LIN {X 0,Y 270.398,Z 235.226,A -85,B 0,C 180,E1 -18840.758,E2 -18840.758} C_VEL
LIN {X 0,Y 266.71,Z 211.064,A -85,B 0,C 180,E1 -18842.032,E2 -18842.032} C_VEL
LIN {X 0,Y 265.559,Z 205.31,A -85,B 0,C 180,E1 -18842.384,E2 -18842.384} C_VEL
LIN {X 0,Y 258.994,Z 190.687,A -85,B 0,C 180,E1 -18843.868,E2 -18843.868} C_VEL
LIN {X 0,Y 254.466,Z 181.608,A -85,B 0,C 180,E1 -18844.919,E2 -18844.919} C_VEL
LIN {X 0,Y 253.32,Z 178.871,A -85,B 0,C 180,E1 -18845.269,E2 -18845.269} C_VEL
LIN {X 0,Y 251.431,Z 171.126,A -85,B 0,C 180,E1 -18848.495,E2 -18848.495} C_VEL
LIN {X 0,Y 249.031,Z 162.462,A -85,B 0,C 180,E1 -18852.416,E2 -18852.416} C_VEL
LIN {X 0,Y 248.994,Z 162.469,A -85,B 0,C 180,E1 -18857.213,E2 -18857.213} C_VEL
LIN {X 0,Y 249.024,Z 162.467,A -85,B 0,C 180,E1 -18861.619,E2 -18861.619} C_VEL
LIN {X 0,Y 249.046,Z 162.465,A -85,B 0,C 180,E1 -18865.64,E2 -18865.64} C_VEL
LIN {X 0,Y 249.005,Z 162.467,A -85,B 0,C 180,E1 -18869.467,E2 -18869.467} C_VEL
LIN {X 0,Y 249.038,Z 162.464,A -85,B 0,C 180,E1 -18873.158,E2 -18873.158} C_VEL
LIN {X 0,Y 249.054,Z 162.46,A -85,B 0,C 180,E1 -18876.73,E2 -18876.73} C_VEL
LIN {X 0,Y 249.044,Z 162.449,A -85,B 0,C 180,E1 -18880.206,E2 -18880.206} C_VEL
LIN {X 0,Y 249.161,Z 162.447,A -85,B 0,C 180,E1 -18883.616,E2 -18883.616} C_VEL
LIN {X 0,Y 249.218,Z 162.442,A -85,B 0,C 180,E1 -18888.615,E2 -18888.615} C_VEL
LIN {X 0,Y 249.405,Z 162.403,A -85,B 0,C 180,E1 -18891.9,E2 -18891.9} C_VEL
LIN {X 0,Y 249.253,Z 162.436,A -85,B 0,C 180,E1 -18895.148,E2 -18895.148} C_VEL
LIN {X 0,Y 249.648,Z 162.378,A -85,B 0,C 180,E1 -18898.387,E2 -18898.387} C_VEL
LIN {X 0,Y 249.656,Z 162.378,A -85,B 0,C 180,E1 -18901.613,E2 -18901.613} C_VEL
LIN {X 0,Y 249.423,Z 162.413,A -85,B 0,C 180,E1 -18906.55,E2 -18906.55} C_VEL
LIN {X 0,Y 249.346,Z 162.414,A -85,B 0,C 180,E1 -18909.737,E2 -18909.737} C_VEL
LIN {X 0,Y 249.174,Z 162.433,A -85,B 0,C 180,E1 -18914.706,E2 -18914.706} C_VEL
LIN {X 0,Y 249.098,Z 162.452,A -85,B 0,C 180,E1 -18918.081,E2 -18918.081} C_VEL
LIN {X 0,Y 249.049,Z 162.463,A -85,B 0,C 180,E1 -18921.522,E2 -18921.522} C_VEL
LIN {X 0,Y 249.09,Z 162.452,A -85,B 0,C 180,E1 -18925.46,E2 -18925.46} C_VEL
LIN {X 0,Y 249.043,Z 162.455,A -85,B 0,C 180,E1 -18928.975,E2 -18928.975} C_VEL
LIN {X 0,Y 249.031,Z 162.458,A -85,B 0,C 180,E1 -18932.426,E2 -18932.426} C_VEL
LIN {X 0,Y 249.034,Z 162.457,A -85,B 0,C 180,E1 -18936.345,E2 -18936.345} C_VEL
LIN {X 0,Y 248.996,Z 162.444,A -85,B 0,C 180,E1 -18940.481,E2 -18940.481} C_VEL
LIN {X 0,Y 249.013,Z 162.453,A -85,B 0,C 180,E1 -18942.792,E2 -18942.792} C_VEL
LIN {X 0,Y 249.02,Z 162.464,A -85,B 0,C 180,E1 -18947.362,E2 -18947.362} C_VEL
LIN {X 0,Y 249.001,Z 162.471,A -85,B 0,C 180,E1 -18949.121,E2 -18949.121} C_VEL
LIN {X 0,Y 249.95,Z 165.205,A -85,B 0,C 180,E1 -18949.392,E2 -18949.392} C_VEL
LIN {X 0,Y 251.706,Z 167.591,A -85,B 0,C 180,E1 -18949.79,E2 -18949.79} C_VEL
LIN {X 0,Y 260.09,Z 181.406,A -85,B 0,C 180,E1 -18951.672,E2 -18951.672} C_VEL
LIN {X 0,Y 267.579,Z 196.726,A -85,B 0,C 180,E1 -18953.313,E2 -18953.313} C_VEL
LIN {X 0,Y 271.539,Z 205.911,A -85,B 0,C 180,E1 -18954.166,E2 -18954.166} C_VEL
LIN {X 0,Y 269.168,Z 267.873,A -85,B 0,C 180,E1 -18955.806,E2 -18955.806} C_VEL
LIN {X 0,Y 268.098,Z 281.069,A -85,B 0,C 180,E1 -18956.441,E2 -18956.441} C_VEL
LIN {X 0,Y 266.619,Z 293.102,A -85,B 0,C 180,E1 -18957.291,E2 -18957.291} C_VEL
LIN {X 0,Y 264.901,Z 304.551,A -85,B 0,C 180,E1 -18958.399,E2 -18958.399} C_VEL
LIN {X 0,Y 262.647,Z 316.276,A -85,B 0,C 180,E1 -18959.885,E2 -18959.885} C_VEL
LIN {X 0,Y 260.185,Z 326.779,A -85,B 0,C 180,E1 -18961.569,E2 -18961.569} C_VEL
LIN {X 0,Y 258.084,Z 335.342,A -85,B 0,C 180,E1 -18963.299,E2 -18963.299} C_VEL
LIN {X 0,Y 255.942,Z 343.505,A -85,B 0,C 180,E1 -18965.332,E2 -18965.332} C_VEL
LIN {X 0,Y 253.727,Z 350.862,A -85,B 0,C 180,E1 -18967.612,E2 -18967.612} C_VEL
LIN {X 0,Y 251.511,Z 357.887,A -85,B 0,C 180,E1 -18970.407,E2 -18970.407} C_VEL
LIN {X 0,Y 249.934,Z 362.747,A -85,B 0,C 180,E1 -18972.954,E2 -18972.954} C_VEL
LIN {X 0,Y 248.859,Z 366.06,A -85,B 0,C 180,E1 -18975.274,E2 -18975.274} C_VEL
LIN {X 0,Y 248.197,Z 367.857,A -85,B 0,C 180,E1 -18976.906,E2 -18976.906} C_VEL
LIN {X 0,Y 247.456,Z 370.137,A -85,B 0,C 180,E1 -18980.187,E2 -18980.187} C_VEL
LIN {X 0,Y 247.288,Z 370.694,A -85,B 0,C 180,E1 -18981.829,E2 -18981.829} C_VEL
LIN {X 0,Y 247.235,Z 370.759,A -85,B 0,C 180,E1 -18984.229,E2 -18984.229} C_VEL
LIN {X 0,Y 247.141,Z 369.941,A -85,B 0,C 180,E1 -18986.738,E2 -18986.738} C_VEL
LIN {X 0,Y 247.152,Z 368.924,A -85,B 0,C 180,E1 -18988.369,E2 -18988.369} C_VEL
LIN {X 0,Y 247.262,Z 367.49,A -85,B 0,C 180,E1 -18989.999,E2 -18989.999} C_VEL
LIN {X 0,Y 247.779,Z 364.536,A -85,B 0,C 180,E1 -18992.437,E2 -18992.437} C_VEL
LIN {X 0,Y 248.415,Z 360.557,A -85,B 0,C 180,E1 -18994.867,E2 -18994.867} C_VEL
LIN {X 0,Y 249.433,Z 355.427,A -85,B 0,C 180,E1 -18997.283,E2 -18997.283} C_VEL
LIN {X 0,Y 250.574,Z 348.992,A -85,B 0,C 180,E1 -18999.687,E2 -18999.687} C_VEL
LIN {X 0,Y 252.341,Z 340.966,A -85,B 0,C 180,E1 -19002.055,E2 -19002.055} C_VEL
LIN {X 0,Y 253.91,Z 332.787,A -85,B 0,C 180,E1 -19004.014,E2 -19004.014} C_VEL
LIN {X 0,Y 255.731,Z 322.787,A -85,B 0,C 180,E1 -19005.95,E2 -19005.95} C_VEL
LIN {X 0,Y 257.53,Z 311.457,A -85,B 0,C 180,E1 -19007.672,E2 -19007.672} C_VEL
LIN {X 0,Y 259.116,Z 300.335,A -85,B 0,C 180,E1 -19008.993,E2 -19008.993} C_VEL
LIN {X 0,Y 260.379,Z 287.896,A -85,B 0,C 180,E1 -19010.128,E2 -19010.128} C_VEL
LIN {X 0,Y 261.415,Z 274.564,A -85,B 0,C 180,E1 -19010.969,E2 -19010.969} C_VEL
LIN {X 0,Y 262.065,Z 261.42,A -85,B 0,C 180,E1 -19011.481,E2 -19011.481} C_VEL
LIN {X 0,Y 264.04,Z 197.022,A -85,B 0,C 180,E1 -19013.187,E2 -19013.187} C_VEL
LIN {X 0,Y 258.122,Z 181.409,A -85,B 0,C 180,E1 -19014.316,E2 -19014.316} C_VEL
LIN {X 0,Y 251.947,Z 168.721,A -85,B 0,C 180,E1 -19015.449,E2 -19015.449} C_VEL
LIN {X 0,Y 249.298,Z 163.437,A -85,B 0,C 180,E1 -19015.951,E2 -19015.951} C_VEL
LIN {X 0,Y 249.084,Z 162.459,A -85,B 0,C 180,E1 -19016.07,E2 -19016.07} C_VEL
LIN {X 0,Y 249.082,Z 162.456,A -85,B 0,C 180,E1 -19018.992,E2 -19018.992} C_VEL
LIN {X 0,Y 249.034,Z 162.462,A -85,B 0,C 180,E1 -19022.423,E2 -19022.423} C_VEL
LIN {X 0,Y 249.064,Z 162.458,A -85,B 0,C 180,E1 -19026.337,E2 -19026.337} C_VEL
LIN {X 0,Y 249.002,Z 162.466,A -85,B 0,C 180,E1 -19030.476,E2 -19030.476} C_VEL
LIN {X 0,Y 248.998,Z 162.467,A -85,B 0,C 180,E1 -19034.877,E2 -19034.877} C_VEL
LIN {X 0,Y 249.011,Z 162.463,A -85,B 0,C 180,E1 -19037.361,E2 -19037.361} C_VEL
LIN {X 0,Y 249.038,Z 162.46,A -85,B 0,C 180,E1 -19042.198,E2 -19042.198} C_VEL
LIN {X 0,Y 249.037,Z 162.464,A -85,B 0,C 180,E1 -19045.638,E2 -19045.638} C_VEL
LIN {X 0,Y 249.039,Z 162.465,A -85,B 0,C 180,E1 -19049.471,E2 -19049.471} C_VEL
LIN {X 0,Y 249.052,Z 162.456,A -85,B 0,C 180,E1 -19053.159,E2 -19053.159} C_VEL
LIN {X 0,Y 249.05,Z 162.46,A -85,B 0,C 180,E1 -19056.729,E2 -19056.729} C_VEL
LIN {X 0,Y 249.069,Z 162.458,A -85,B 0,C 180,E1 -19060.208,E2 -19060.208} C_VEL
LIN {X 0,Y 249.168,Z 162.441,A -85,B 0,C 180,E1 -19063.617,E2 -19063.617} C_VEL
LIN {X 0,Y 249.221,Z 162.439,A -85,B 0,C 180,E1 -19068.615,E2 -19068.615} C_VEL
LIN {X 0,Y 249.407,Z 162.4,A -85,B 0,C 180,E1 -19071.9,E2 -19071.9} C_VEL
LIN {X 0,Y 249.247,Z 162.411,A -85,B 0,C 180,E1 -19075.147,E2 -19075.147} C_VEL
LIN {X 0,Y 249.645,Z 162.383,A -85,B 0,C 180,E1 -19078.387,E2 -19078.387} C_VEL
LIN {X 0,Y 249.646,Z 162.385,A -85,B 0,C 180,E1 -19081.613,E2 -19081.613} C_VEL
LIN {X 0,Y 249.386,Z 162.415,A -85,B 0,C 180,E1 -19087.553,E2 -19087.553} C_VEL
LIN {X 0,Y 248.706,Z 162.507,A -85,B 0,C 180,E1 -19088.899,E2 -19088.899} C_VEL
LIN {X 0,Y 245.74,Z 162.873,A -85,B 0,C 180,E1 -19091.09,E2 -19091.09} C_VEL
LIN {X 0,Y 243.227,Z 163.188,A -85,B 0,C 180,E1 -19092.875,E2 -19092.875} C_VEL
LIN {X 0,Y 242.172,Z 163.32,A -85,B 0,C 180,E1 -19094.263,E2 -19094.263} C_VEL
LIN {X 0,Y 242.099,Z 163.326,A -85,B 0,C 180,E1 -19094.734,E2 -19094.734} C_VEL
LIN {X 0,Y 242.033,Z 163.341,A -85,B 0,C 180,E1 -19098.627,E2 -19098.627} C_VEL
LIN {X 0,Y 241.995,Z 163.343,A -85,B 0,C 180,E1 -19102.182,E2 -19102.182} C_VEL
LIN {X 0,Y 242.059,Z 163.334,A -85,B 0,C 180,E1 -19105.839,E2 -19105.839} C_VEL
LIN {X 0,Y 241.996,Z 163.342,A -85,B 0,C 180,E1 -19109.585,E2 -19109.585} C_VEL
LIN {X 0,Y 241.973,Z 163.345,A -85,B 0,C 180,E1 -19113.494,E2 -19113.494} C_VEL
LIN {X 0,Y 241.982,Z 163.344,A -85,B 0,C 180,E1 -19117.583,E2 -19117.583} C_VEL
LIN {X 0,Y 241.931,Z 163.351,A -85,B 0,C 180,E1 -19121.924,E2 -19121.924} C_VEL
LIN {X 0,Y 241.928,Z 163.347,A -85,B 0,C 180,E1 -19126.573,E2 -19126.573} C_VEL
LIN {X 0,Y 241.952,Z 163.347,A -85,B 0,C 180,E1 -19130.283,E2 -19130.283} C_VEL
LIN {X 0,Y 242.037,Z 163.517,A -85,B 0,C 180,E1 -19132.235,E2 -19132.235} C_VEL
LIN {X 0,Y 244.204,Z 172.335,A -85,B 0,C 180,E1 -19135.78,E2 -19135.78} C_VEL
LIN {X 0,Y 245.763,Z 179.777,A -85,B 0,C 180,E1 -19138.518,E2 -19138.518} C_VEL
LIN {X 0,Y 251.548,Z 194.496,A -85,B 0,C 180,E1 -19139.711,E2 -19139.711} C_VEL
LIN {X 0,Y 254.766,Z 216.953,A -85,B 0,C 180,E1 -19140.788,E2 -19140.788} C_VEL
LIN {X 0,Y 256.54,Z 232.58,A -85,B 0,C 180,E1 -19141.465,E2 -19141.465} C_VEL
LIN {X 0,Y 254.785,Z 288.121,A -85,B 0,C 180,E1 -19143.004,E2 -19143.004} C_VEL
LIN {X 0,Y 253.886,Z 301.362,A -85,B 0,C 180,E1 -19143.659,E2 -19143.659} C_VEL
LIN {X 0,Y 252.596,Z 312.538,A -85,B 0,C 180,E1 -19144.455,E2 -19144.455} C_VEL
LIN {X 0,Y 250.923,Z 324.371,A -85,B 0,C 180,E1 -19145.601,E2 -19145.601} C_VEL
LIN {X 0,Y 249.17,Z 335.145,A -85,B 0,C 180,E1 -19146.963,E2 -19146.963} C_VEL
LIN {X 0,Y 247.068,Z 346.126,A -85,B 0,C 180,E1 -19148.737,E2 -19148.737} C_VEL
LIN {X 0,Y 245.138,Z 356.346,A -85,B 0,C 180,E1 -19150.838,E2 -19150.838} C_VEL
LIN {X 0,Y 243.792,Z 364.08,A -85,B 0,C 180,E1 -19152.815,E2 -19152.815} C_VEL
LIN {X 0,Y 242.455,Z 370.774,A -85,B 0,C 180,E1 -19154.879,E2 -19154.879} C_VEL
LIN {X 0,Y 241.155,Z 377.362,A -85,B 0,C 180,E1 -19157.377,E2 -19157.377} C_VEL
LIN {X 0,Y 240.425,Z 382.612,A -85,B 0,C 180,E1 -19159.9,E2 -19159.9} C_VEL
LIN {X 0,Y 240.024,Z 386.683,A -85,B 0,C 180,E1 -19162.43,E2 -19162.43} C_VEL
LIN {X 0,Y 239.92,Z 389.691,A -85,B 0,C 180,E1 -19164.96,E2 -19164.96} C_VEL
LIN {X 0,Y 239.918,Z 391.144,A -85,B 0,C 180,E1 -19166.643,E2 -19166.643} C_VEL
LIN {X 0,Y 239.991,Z 392.169,A -85,B 0,C 180,E1 -19168.323,E2 -19168.323} C_VEL
LIN {X 0,Y 240.018,Z 392.796,A -85,B 0,C 180,E1 -19170.002,E2 -19170.002} C_VEL
LIN {X 0,Y 239.971,Z 393.027,A -85,B 0,C 180,E1 -19171.68,E2 -19171.68} C_VEL
LIN {X 0,Y 239.846,Z 392.272,A -85,B 0,C 180,E1 -19174.948,E2 -19174.948} C_VEL
LIN {X 0,Y 239.899,Z 391.228,A -85,B 0,C 180,E1 -19176.731,E2 -19176.731} C_VEL
LIN {X 0,Y 240.146,Z 389.843,A -85,B 0,C 180,E1 -19178.416,E2 -19178.416} C_VEL
LIN {X 0,Y 240.77,Z 386.934,A -85,B 0,C 180,E1 -19180.939,E2 -19180.939} C_VEL
LIN {X 0,Y 241.714,Z 383.006,A -85,B 0,C 180,E1 -19183.452,E2 -19183.452} C_VEL
LIN {X 0,Y 243.32,Z 377.97,A -85,B 0,C 180,E1 -19185.927,E2 -19185.927} C_VEL
LIN {X 0,Y 245.241,Z 371.662,A -85,B 0,C 180,E1 -19188.376,E2 -19188.376} C_VEL
LIN {X 0,Y 247.394,Z 363.783,A -85,B 0,C 180,E1 -19190.801,E2 -19190.801} C_VEL
LIN {X 0,Y 249.742,Z 355.777,A -85,B 0,C 180,E1 -19192.765,E2 -19192.765} C_VEL
LIN {X 0,Y 252.414,Z 346.028,A -85,B 0,C 180,E1 -19194.687,E2 -19194.687} C_VEL
LIN {X 0,Y 255.143,Z 335.198,A -85,B 0,C 180,E1 -19196.371,E2 -19196.371} C_VEL
LIN {X 0,Y 257.365,Z 324.63,A -85,B 0,C 180,E1 -19197.661,E2 -19197.661} C_VEL
LIN {X 0,Y 259.68,Z 311.918,A -85,B 0,C 180,E1 -19198.822,E2 -19198.822} C_VEL
LIN {X 0,Y 261.438,Z 299.188,A -85,B 0,C 180,E1 -19199.658,E2 -19199.658} C_VEL
LIN {X 0,Y 262.469,Z 286.951,A -85,B 0,C 180,E1 -19200.193,E2 -19200.193} C_VEL
LIN {X 0,Y 264.433,Z 236.333,A -85,B 0,C 180,E1 -19201.554,E2 -19201.554} C_VEL
LIN {X 0,Y 260.963,Z 213.15,A -85,B 0,C 180,E1 -19202.816,E2 -19202.816} C_VEL
LIN {X 0,Y 259.786,Z 207.659,A -85,B 0,C 180,E1 -19203.178,E2 -19203.178} C_VEL
LIN {X 0,Y 252.386,Z 191.247,A -85,B 0,C 180,E1 -19204.937,E2 -19204.937} C_VEL
LIN {X 0,Y 247.472,Z 181.709,A -85,B 0,C 180,E1 -19206.138,E2 -19206.138} C_VEL
LIN {X 0,Y 246.043,Z 178.541,A -85,B 0,C 180,E1 -19206.547,E2 -19206.547} C_VEL
LIN {X 0,Y 244.236,Z 171.448,A -85,B 0,C 180,E1 -19209.661,E2 -19209.661} C_VEL
LIN {X 0,Y 241.934,Z 163.348,A -85,B 0,C 180,E1 -19213.573,E2 -19213.573} C_VEL
LIN {X 0,Y 241.925,Z 163.351,A -85,B 0,C 180,E1 -19218.075,E2 -19218.075} C_VEL
LIN {X 0,Y 241.988,Z 163.343,A -85,B 0,C 180,E1 -19222.418,E2 -19222.418} C_VEL
LIN {X 0,Y 241.982,Z 163.344,A -85,B 0,C 180,E1 -19226.508,E2 -19226.508} C_VEL
LIN {X 0,Y 241.98,Z 163.345,A -85,B 0,C 180,E1 -19230.613,E2 -19230.613} C_VEL
LIN {X 0,Y 242.035,Z 163.333,A -85,B 0,C 180,E1 -19234.179,E2 -19234.179} C_VEL
LIN {X 0,Y 241.995,Z 163.34,A -85,B 0,C 180,E1 -19238.335,E2 -19238.335} C_VEL
LIN {X 0,Y 242.108,Z 163.326,A -85,B 0,C 180,E1 -19243.325,E2 -19243.325} C_VEL
LIN {X 0,Y 242.152,Z 163.321,A -85,B 0,C 180,E1 -19248.278,E2 -19248.278} C_VEL
LIN {X 0,Y 242.36,Z 163.28,A -85,B 0,C 180,E1 -19251.663,E2 -19251.663} C_VEL
LIN {X 0,Y 242.392,Z 163.289,A -85,B 0,C 180,E1 -19253.34,E2 -19253.34} C_VEL
LIN {X 0,Y 242.608,Z 163.254,A -85,B 0,C 180,E1 -19258.34,E2 -19258.34} C_VEL
LIN {X 0,Y 242.616,Z 163.254,A -85,B 0,C 180,E1 -19261.66,E2 -19261.66} C_VEL
LIN {X 0,Y 242.398,Z 163.289,A -85,B 0,C 180,E1 -19266.66,E2 -19266.66} C_VEL
LIN {X 0,Y 242.269,Z 163.299,A -85,B 0,C 180,E1 -19270.024,E2 -19270.024} C_VEL
LIN {X 0,Y 242.124,Z 163.313,A -85,B 0,C 180,E1 -19275.144,E2 -19275.144} C_VEL
LIN {X 0,Y 242.034,Z 163.327,A -85,B 0,C 180,E1 -19278.627,E2 -19278.627} C_VEL
LIN {X 0,Y 241.991,Z 163.341,A -85,B 0,C 180,E1 -19282.182,E2 -19282.182} C_VEL
LIN {X 0,Y 242.036,Z 163.334,A -85,B 0,C 180,E1 -19285.821,E2 -19285.821} C_VEL
LIN {X 0,Y 241.973,Z 163.338,A -85,B 0,C 180,E1 -19289.588,E2 -19289.588} C_VEL
LIN {X 0,Y 241.983,Z 163.337,A -85,B 0,C 180,E1 -19293.493,E2 -19293.493} C_VEL
LIN {X 0,Y 241.991,Z 163.34,A -85,B 0,C 180,E1 -19297.582,E2 -19297.582} C_VEL
LIN {X 0,Y 241.938,Z 163.324,A -85,B 0,C 180,E1 -19301.923,E2 -19301.923} C_VEL
LIN {X 0,Y 241.938,Z 163.35,A -85,B 0,C 180,E1 -19306.571,E2 -19306.571} C_VEL
LIN {X 0,Y 241.962,Z 163.343,A -85,B 0,C 180,E1 -19307.816,E2 -19307.816} C_VEL
LIN {X 0,Y 242.91,Z 166.061,A -85,B 0,C 180,E1 -19308.105,E2 -19308.105} C_VEL
LIN {X 0,Y 244.803,Z 168.669,A -85,B 0,C 180,E1 -19308.566,E2 -19308.566} C_VEL
LIN {X 0,Y 253.616,Z 182.897,A -85,B 0,C 180,E1 -19310.658,E2 -19310.658} C_VEL
LIN {X 0,Y 258.598,Z 192.44,A -85,B 0,C 180,E1 -19311.804,E2 -19311.804} C_VEL
LIN {X 0,Y 265.417,Z 207.578,A -85,B 0,C 180,E1 -19313.344,E2 -19313.344} C_VEL
LIN {X 0,Y 265.285,Z 215.569,A -85,B 0,C 180,E1 -19313.581,E2 -19313.581} C_VEL
LIN {X 0,Y 263.163,Z 268.09,A -85,B 0,C 180,E1 -19314.999,E2 -19314.999} C_VEL
LIN {X 0,Y 262.004,Z 281.688,A -85,B 0,C 180,E1 -19315.665,E2 -19315.665} C_VEL
LIN {X 0,Y 260.461,Z 293.792,A -85,B 0,C 180,E1 -19316.544,E2 -19316.544} C_VEL
LIN {X 0,Y 258.721,Z 304.882,A -85,B 0,C 180,E1 -19317.644,E2 -19317.644} C_VEL
LIN {X 0,Y 256.473,Z 316.095,A -85,B 0,C 180,E1 -19319.082,E2 -19319.082} C_VEL
LIN {X 0,Y 253.93,Z 326.686,A -85,B 0,C 180,E1 -19320.802,E2 -19320.802} C_VEL
LIN {X 0,Y 251.679,Z 335.319,A -85,B 0,C 180,E1 -19322.563,E2 -19322.563} C_VEL
LIN {X 0,Y 249.574,Z 342.981,A -85,B 0,C 180,E1 -19324.487,E2 -19324.487} C_VEL
LIN {X 0,Y 247.54,Z 349.798,A -85,B 0,C 180,E1 -19326.578,E2 -19326.578} C_VEL
LIN {X 0,Y 245.375,Z 356.227,A -85,B 0,C 180,E1 -19329.02,E2 -19329.02} C_VEL
LIN {X 0,Y 243.658,Z 361.302,A -85,B 0,C 180,E1 -19331.5,E2 -19331.5} C_VEL
LIN {X 0,Y 242.263,Z 365.227,A -85,B 0,C 180,E1 -19334.001,E2 -19334.001} C_VEL
LIN {X 0,Y 241.24,Z 368.108,A -85,B 0,C 180,E1 -19336.521,E2 -19336.521} C_VEL
LIN {X 0,Y 240.407,Z 370.424,A -85,B 0,C 180,E1 -19339.896,E2 -19339.896} C_VEL
LIN {X 0,Y 240.172,Z 371.171,A -85,B 0,C 180,E1 -19343.277,E2 -19343.277} C_VEL
LIN {X 0,Y 240.077,Z 370.927,A -85,B 0,C 180,E1 -19344.96,E2 -19344.96} C_VEL
LIN {X 0,Y 240.055,Z 370.304,A -85,B 0,C 180,E1 -19346.642,E2 -19346.642} C_VEL
LIN {X 0,Y 240.077,Z 369.302,A -85,B 0,C 180,E1 -19348.321,E2 -19348.321} C_VEL
LIN {X 0,Y 240.18,Z 367.899,A -85,B 0,C 180,E1 -19349.998,E2 -19349.998} C_VEL
LIN {X 0,Y 240.692,Z 364.974,A -85,B 0,C 180,E1 -19352.509,E2 -19352.509} C_VEL
LIN {X 0,Y 241.358,Z 361.028,A -85,B 0,C 180,E1 -19355.01,E2 -19355.01} C_VEL
LIN {X 0,Y 242.423,Z 355.942,A -85,B 0,C 180,E1 -19357.494,E2 -19357.494} C_VEL
LIN {X 0,Y 243.608,Z 349.555,A -85,B 0,C 180,E1 -19359.966,E2 -19359.966} C_VEL
LIN {X 0,Y 245.437,Z 341.577,A -85,B 0,C 180,E1 -19362.4,E2 -19362.4} C_VEL
LIN {X 0,Y 247.078,Z 333.455,A -85,B 0,C 180,E1 -19364.41,E2 -19364.41} C_VEL
LIN {X 0,Y 248.946,Z 323.547,A -85,B 0,C 180,E1 -19366.396,E2 -19366.396} C_VEL
LIN {X 0,Y 250.823,Z 312.331,A -85,B 0,C 180,E1 -19368.161,E2 -19368.161} C_VEL
LIN {X 0,Y 252.476,Z 301.338,A -85,B 0,C 180,E1 -19369.512,E2 -19369.512} C_VEL
LIN {X 0,Y 253.792,Z 289.172,A -85,B 0,C 180,E1 -19370.674,E2 -19370.674} C_VEL
LIN {X 0,Y 254.859,Z 276.299,A -85,B 0,C 180,E1 -19371.535,E2 -19371.535} C_VEL
LIN {X 0,Y 255.591,Z 262.578,A -85,B 0,C 180,E1 -19372.107,E2 -19372.107} C_VEL
LIN {X 0,Y 257.602,Z 198.497,A -85,B 0,C 180,E1 -19373.851,E2 -19373.851} C_VEL
LIN {X 0,Y 251.964,Z 183.792,A -85,B 0,C 180,E1 -19374.969,E2 -19374.969} C_VEL
LIN {X 0,Y 244.995,Z 169.7,A -85,B 0,C 180,E1 -19376.304,E2 -19376.304} C_VEL
LIN {X 0,Y 242.27,Z 164.505,A -85,B 0,C 180,E1 -19376.842,E2 -19376.842} C_VEL
LIN {X 0,Y 242.031,Z 163.337,A -85,B 0,C 180,E1 -19376.936,E2 -19376.936} C_VEL
LIN {X 0,Y 242.029,Z 163.335,A -85,B 0,C 180,E1 -19379.578,E2 -19379.578} C_VEL
LIN {X 0,Y 241.989,Z 163.34,A -85,B 0,C 180,E1 -19383.489,E2 -19383.489} C_VEL
LIN {X 0,Y 241.995,Z 163.339,A -85,B 0,C 180,E1 -19387.578,E2 -19387.578} C_VEL
LIN {X 0,Y 241.933,Z 163.348,A -85,B 0,C 180,E1 -19391.92,E2 -19391.92} C_VEL
LIN {X 0,Y 241.929,Z 163.346,A -85,B 0,C 180,E1 -19396.57,E2 -19396.57} C_VEL
LIN {X 0,Y 241.951,Z 163.346,A -85,B 0,C 180,E1 -19400.279,E2 -19400.279} C_VEL
LIN {X 0,Y 241.982,Z 163.342,A -85,B 0,C 180,E1 -19404.488,E2 -19404.488} C_VEL
LIN {X 0,Y 241.965,Z 163.343,A -85,B 0,C 180,E1 -19408.478,E2 -19408.478} C_VEL
LIN {X 0,Y 241.984,Z 163.335,A -85,B 0,C 180,E1 -19412.309,E2 -19412.309} C_VEL
LIN {X 0,Y 242.03,Z 163.336,A -85,B 0,C 180,E1 -19416.013,E2 -19416.013} C_VEL
LIN {X 0,Y 242.008,Z 163.337,A -85,B 0,C 180,E1 -19419.605,E2 -19419.605} C_VEL
LIN {X 0,Y 242.107,Z 163.323,A -85,B 0,C 180,E1 -19423.315,E2 -19423.315} C_VEL
LIN {X 0,Y 242.155,Z 163.319,A -85,B 0,C 180,E1 -19428.278,E2 -19428.278} C_VEL
LIN {X 0,Y 242.361,Z 163.277,A -85,B 0,C 180,E1 -19431.663,E2 -19431.663} C_VEL
LIN {X 0,Y 242.385,Z 163.26,A -85,B 0,C 180,E1 -19433.34,E2 -19433.34} C_VEL
LIN {X 0,Y 242.605,Z 163.259,A -85,B 0,C 180,E1 -19438.34,E2 -19438.34} C_VEL
LIN {X 0,Y 242.606,Z 163.262,A -85,B 0,C 180,E1 -19441.66,E2 -19441.66} C_VEL
LIN {X 0,Y 242.345,Z 163.293,A -85,B 0,C 180,E1 -19447.548,E2 -19447.548} C_VEL
LIN {X 0,Y 242.252,Z 163.309,A -85,B 0,C 180,E1 -19450.024,E2 -19450.024} C_VEL
LIN {X 0,Y 242.099,Z 163.326,A -85,B 0,C 180,E1 -19454.734,E2 -19454.734} C_VEL
LIN {X 0,Y 241.466,Z 163.409,A -85,B 0,C 180,E1 -19456.122,E2 -19456.122} C_VEL
LIN {X 0,Y 238.616,Z 163.766,A -85,B 0,C 180,E1 -19458.384,E2 -19458.384} C_VEL
LIN {X 0,Y 236.151,Z 164.072,A -85,B 0,C 180,E1 -19460.228,E2 -19460.228} C_VEL
LIN {X 0,Y 235.062,Z 164.206,A -85,B 0,C 180,E1 -19461.659,E2 -19461.659} C_VEL
LIN {X 0,Y 234.958,Z 164.219,A -85,B 0,C 180,E1 -19462.145,E2 -19462.145} C_VEL
LIN {X 0,Y 234.956,Z 164.223,A -85,B 0,C 180,E1 -19466.659,E2 -19466.659} C_VEL
LIN {X 0,Y 234.913,Z 164.228,A -85,B 0,C 180,E1 -19470.57,E2 -19470.57} C_VEL
LIN {X 0,Y 234.923,Z 164.226,A -85,B 0,C 180,E1 -19474.639,E2 -19474.639} C_VEL
LIN {X 0,Y 234.935,Z 164.222,A -85,B 0,C 180,E1 -19478.946,E2 -19478.946} C_VEL
LIN {X 0,Y 234.881,Z 164.228,A -85,B 0,C 180,E1 -19483.487,E2 -19483.487} C_VEL
LIN {X 0,Y 234.881,Z 164.225,A -85,B 0,C 180,E1 -19486.516,E2 -19486.516} C_VEL
LIN {X 0,Y 234.963,Z 164.296,A -85,B 0,C 180,E1 -19491.451,E2 -19491.451} C_VEL
LIN {X 0,Y 237.196,Z 173.334,A -85,B 0,C 180,E1 -19495.227,E2 -19495.227} C_VEL
LIN {X 0,Y 238.472,Z 179.327,A -85,B 0,C 180,E1 -19497.529,E2 -19497.529} C_VEL
LIN {X 0,Y 245.438,Z 196.678,A -85,B 0,C 180,E1 -19499.029,E2 -19499.029} C_VEL
LIN {X 0,Y 248.322,Z 216.781,A -85,B 0,C 180,E1 -19500.032,E2 -19500.032} C_VEL
LIN {X 0,Y 250.179,Z 234.602,A -85,B 0,C 180,E1 -19500.816,E2 -19500.816} C_VEL
LIN {X 0,Y 248.329,Z 288.491,A -85,B 0,C 180,E1 -19502.347,E2 -19502.347} C_VEL
LIN {X 0,Y 247.366,Z 301.6,A -85,B 0,C 180,E1 -19503.021,E2 -19503.021} C_VEL
LIN {X 0,Y 246.047,Z 312.647,A -85,B 0,C 180,E1 -19503.838,E2 -19503.838} C_VEL
LIN {X 0,Y 244.462,Z 323.498,A -85,B 0,C 180,E1 -19504.912,E2 -19504.912} C_VEL
LIN {X 0,Y 242.616,Z 334.378,A -85,B 0,C 180,E1 -19506.303,E2 -19506.303} C_VEL
LIN {X 0,Y 240.73,Z 344.388,A -85,B 0,C 180,E1 -19507.923,E2 -19507.923} C_VEL
LIN {X 0,Y 238.784,Z 353.578,A -85,B 0,C 180,E1 -19509.769,E2 -19509.769} C_VEL
LIN {X 0,Y 237.184,Z 362.309,A -85,B 0,C 180,E1 -19511.961,E2 -19511.961} C_VEL
LIN {X 0,Y 235.549,Z 370.257,A -85,B 0,C 180,E1 -19514.425,E2 -19514.425} C_VEL
LIN {X 0,Y 234.203,Z 376.882,A -85,B 0,C 180,E1 -19516.995,E2 -19516.995} C_VEL
LIN {X 0,Y 233.411,Z 382.166,A -85,B 0,C 180,E1 -19519.594,E2 -19519.594} C_VEL
LIN {X 0,Y 232.974,Z 386.266,A -85,B 0,C 180,E1 -19522.2,E2 -19522.2} C_VEL
LIN {X 0,Y 232.842,Z 389.408,A -85,B 0,C 180,E1 -19524.912,E2 -19524.912} C_VEL
LIN {X 0,Y 232.819,Z 390.776,A -85,B 0,C 180,E1 -19526.54,E2 -19526.54} C_VEL
LIN {X 0,Y 232.919,Z 391.816,A -85,B 0,C 180,E1 -19528.273,E2 -19528.273} C_VEL
LIN {X 0,Y 232.946,Z 392.455,A -85,B 0,C 180,E1 -19530.002,E2 -19530.002} C_VEL
LIN {X 0,Y 232.898,Z 392.698,A -85,B 0,C 180,E1 -19531.731,E2 -19531.731} C_VEL
LIN {X 0,Y 232.77,Z 392.081,A -85,B 0,C 180,E1 -19534.884,E2 -19534.884} C_VEL
LIN {X 0,Y 232.82,Z 390.946,A -85,B 0,C 180,E1 -19536.937,E2 -19536.937} C_VEL
LIN {X 0,Y 233.094,Z 389.574,A -85,B 0,C 180,E1 -19538.672,E2 -19538.672} C_VEL
LIN {X 0,Y 233.767,Z 386.69,A -85,B 0,C 180,E1 -19541.271,E2 -19541.271} C_VEL
LIN {X 0,Y 234.787,Z 382.791,A -85,B 0,C 180,E1 -19543.857,E2 -19543.857} C_VEL
LIN {X 0,Y 236.48,Z 377.785,A -85,B 0,C 180,E1 -19546.401,E2 -19546.401} C_VEL
LIN {X 0,Y 238.793,Z 370.492,A -85,B 0,C 180,E1 -19549.271,E2 -19549.271} C_VEL
LIN {X 0,Y 241.198,Z 362.198,A -85,B 0,C 180,E1 -19551.81,E2 -19551.81} C_VEL
LIN {X 0,Y 243.751,Z 353.944,A -85,B 0,C 180,E1 -19553.808,E2 -19553.808} C_VEL
LIN {X 0,Y 246.603,Z 343.874,A -85,B 0,C 180,E1 -19555.762,E2 -19555.762} C_VEL
LIN {X 0,Y 249.443,Z 332.483,A -85,B 0,C 180,E1 -19557.476,E2 -19557.476} C_VEL
LIN {X 0,Y 251.838,Z 321.323,A -85,B 0,C 180,E1 -19558.778,E2 -19558.778} C_VEL
LIN {X 0,Y 254.062,Z 308.847,A -85,B 0,C 180,E1 -19559.864,E2 -19559.864} C_VEL
LIN {X 0,Y 255.777,Z 295.518,A -85,B 0,C 180,E1 -19560.668,E2 -19560.668} C_VEL
LIN {X 0,Y 256.731,Z 282.506,A -85,B 0,C 180,E1 -19561.17,E2 -19561.17} C_VEL
LIN {X 0,Y 258.543,Z 237.621,A -85,B 0,C 180,E1 -19562.378,E2 -19562.378} C_VEL
LIN {X 0,Y 254.711,Z 211.904,A -85,B 0,C 180,E1 -19563.839,E2 -19563.839} C_VEL
LIN {X 0,Y 249.856,Z 200.467,A -85,B 0,C 180,E1 -19565.047,E2 -19565.047} C_VEL
LIN {X 0,Y 243.325,Z 186.984,A -85,B 0,C 180,E1 -19566.711,E2 -19566.711} C_VEL
LIN {X 0,Y 238.785,Z 178.173,A -85,B 0,C 180,E1 -19567.937,E2 -19567.937} C_VEL
LIN {X 0,Y 236.427,Z 169.538,A -85,B 0,C 180,E1 -19572,E2 -19572} C_VEL
LIN {X 0,Y 234.875,Z 164.228,A -85,B 0,C 180,E1 -19574.714,E2 -19574.714} C_VEL
LIN {X 0,Y 234.867,Z 164.229,A -85,B 0,C 180,E1 -19578.829,E2 -19578.829} C_VEL
LIN {X 0,Y 234.928,Z 164.222,A -85,B 0,C 180,E1 -19583.251,E2 -19583.251} C_VEL
LIN {X 0,Y 234.956,Z 164.218,A -85,B 0,C 180,E1 -19587.424,E2 -19587.424} C_VEL
LIN {X 0,Y 234.904,Z 164.222,A -85,B 0,C 180,E1 -19591.4,E2 -19591.4} C_VEL
LIN {X 0,Y 234.956,Z 164.218,A -85,B 0,C 180,E1 -19595.243,E2 -19595.243} C_VEL
LIN {X 0,Y 234.942,Z 164.213,A -85,B 0,C 180,E1 -19598.963,E2 -19598.963} C_VEL
LIN {X 0,Y 235.052,Z 164.205,A -85,B 0,C 180,E1 -19603.098,E2 -19603.098} C_VEL
LIN {X 0,Y 235.084,Z 164.199,A -85,B 0,C 180,E1 -19607.921,E2 -19607.921} C_VEL
LIN {X 0,Y 235.298,Z 164.159,A -85,B 0,C 180,E1 -19611.411,E2 -19611.411} C_VEL
LIN {X 0,Y 235.343,Z 164.166,A -85,B 0,C 180,E1 -19613.14,E2 -19613.14} C_VEL
LIN {X 0,Y 235.567,Z 164.13,A -85,B 0,C 180,E1 -19618.291,E2 -19618.291} C_VEL
LIN {X 0,Y 235.575,Z 164.131,A -85,B 0,C 180,E1 -19621.71,E2 -19621.71} C_VEL
LIN {X 0,Y 235.35,Z 164.166,A -85,B 0,C 180,E1 -19626.86,E2 -19626.86} C_VEL
LIN {X 0,Y 235.215,Z 164.181,A -85,B 0,C 180,E1 -19630.328,E2 -19630.328} C_VEL
LIN {X 0,Y 235.073,Z 164.195,A -85,B 0,C 180,E1 -19635.609,E2 -19635.609} C_VEL
LIN {X 0,Y 234.973,Z 164.203,A -85,B 0,C 180,E1 -19639.209,E2 -19639.209} C_VEL
LIN {X 0,Y 234.941,Z 164.216,A -85,B 0,C 180,E1 -19642.885,E2 -19642.885} C_VEL
LIN {X 0,Y 234.95,Z 164.22,A -85,B 0,C 180,E1 -19646.66,E2 -19646.66} C_VEL
LIN {X 0,Y 234.903,Z 164.225,A -85,B 0,C 180,E1 -19650.572,E2 -19650.572} C_VEL
LIN {X 0,Y 234.931,Z 164.222,A -85,B 0,C 180,E1 -19654.638,E2 -19654.638} C_VEL
LIN {X 0,Y 234.918,Z 164.216,A -85,B 0,C 180,E1 -19658.936,E2 -19658.936} C_VEL
LIN {X 0,Y 234.891,Z 164.222,A -85,B 0,C 180,E1 -19663.486,E2 -19663.486} C_VEL
LIN {X 0,Y 234.912,Z 164.225,A -85,B 0,C 180,E1 -19666.371,E2 -19666.371} C_VEL
LIN {X 0,Y 236.006,Z 167.195,A -85,B 0,C 180,E1 -19666.753,E2 -19666.753} C_VEL
LIN {X 0,Y 237.794,Z 169.484,A -85,B 0,C 180,E1 -19667.214,E2 -19667.214} C_VEL
LIN {X 0,Y 247.041,Z 184.175,A -85,B 0,C 180,E1 -19669.549,E2 -19669.549} C_VEL
LIN {X 0,Y 252.242,Z 193.63,A -85,B 0,C 180,E1 -19670.798,E2 -19670.798} C_VEL
LIN {X 0,Y 258.943,Z 208.37,A -85,B 0,C 180,E1 -19672.39,E2 -19672.39} C_VEL
LIN {X 0,Y 259.633,Z 210.013,A -85,B 0,C 180,E1 -19672.552,E2 -19672.552} C_VEL
LIN {X 0,Y 257.22,Z 268.266,A -85,B 0,C 180,E1 -19674.152,E2 -19674.152} C_VEL
LIN {X 0,Y 256.065,Z 281.47,A -85,B 0,C 180,E1 -19674.803,E2 -19674.803} C_VEL
LIN {X 0,Y 254.383,Z 294.248,A -85,B 0,C 180,E1 -19675.741,E2 -19675.741} C_VEL
LIN {X 0,Y 252.557,Z 305.347,A -85,B 0,C 180,E1 -19676.867,E2 -19676.867} C_VEL
LIN {X 0,Y 250.058,Z 317.212,A -85,B 0,C 180,E1 -19678.434,E2 -19678.434} C_VEL
LIN {X 0,Y 247.428,Z 327.665,A -85,B 0,C 180,E1 -19680.192,E2 -19680.192} C_VEL
LIN {X 0,Y 244.849,Z 337.039,A -85,B 0,C 180,E1 -19682.196,E2 -19682.196} C_VEL
LIN {X 0,Y 242.21,Z 346.06,A -85,B 0,C 180,E1 -19684.659,E2 -19684.659} C_VEL
LIN {X 0,Y 239.754,Z 353.307,A -85,B 0,C 180,E1 -19687.144,E2 -19687.144} C_VEL
LIN {X 0,Y 238.035,Z 358.185,A -85,B 0,C 180,E1 -19689.248,E2 -19689.248} C_VEL
LIN {X 0,Y 236.29,Z 363.047,A -85,B 0,C 180,E1 -19691.89,E2 -19691.89} C_VEL
LIN {X 0,Y 234.993,Z 366.504,A -85,B 0,C 180,E1 -19694.384,E2 -19694.384} C_VEL
LIN {X 0,Y 234.296,Z 368.354,A -85,B 0,C 180,E1 -19696.114,E2 -19696.114} C_VEL
LIN {X 0,Y 233.751,Z 369.736,A -85,B 0,C 180,E1 -19697.849,E2 -19697.849} C_VEL
LIN {X 0,Y 233.158,Z 371.298,A -85,B 0,C 180,E1 -19701.33,E2 -19701.33} C_VEL
LIN {X 0,Y 233.066,Z 371.378,A -85,B 0,C 180,E1 -19704.33,E2 -19704.33} C_VEL
LIN {X 0,Y 232.972,Z 370.666,A -85,B 0,C 180,E1 -19706.54,E2 -19706.54} C_VEL
LIN {X 0,Y 233.004,Z 369.679,A -85,B 0,C 180,E1 -19708.27,E2 -19708.27} C_VEL
LIN {X 0,Y 233.1,Z 368.302,A -85,B 0,C 180,E1 -19709.998,E2 -19709.998} C_VEL
LIN {X 0,Y 233.606,Z 365.404,A -85,B 0,C 180,E1 -19712.585,E2 -19712.585} C_VEL
LIN {X 0,Y 234.301,Z 361.492,A -85,B 0,C 180,E1 -19715.161,E2 -19715.161} C_VEL
LIN {X 0,Y 235.417,Z 356.448,A -85,B 0,C 180,E1 -19717.719,E2 -19717.719} C_VEL
LIN {X 0,Y 236.65,Z 350.115,A -85,B 0,C 180,E1 -19720.262,E2 -19720.262} C_VEL
LIN {X 0,Y 238.546,Z 342.186,A -85,B 0,C 180,E1 -19722.764,E2 -19722.764} C_VEL
LIN {X 0,Y 240.433,Z 333.265,A -85,B 0,C 180,E1 -19725.027,E2 -19725.027} C_VEL
LIN {X 0,Y 242.391,Z 323.178,A -85,B 0,C 180,E1 -19727.07,E2 -19727.07} C_VEL
LIN {X 0,Y 244.365,Z 311.787,A -85,B 0,C 180,E1 -19728.876,E2 -19728.876} C_VEL
LIN {X 0,Y 246.088,Z 300.589,A -85,B 0,C 180,E1 -19730.258,E2 -19730.258} C_VEL
LIN {X 0,Y 247.332,Z 289.235,A -85,B 0,C 180,E1 -19731.348,E2 -19731.348} C_VEL
LIN {X 0,Y 248.44,Z 276.221,A -85,B 0,C 180,E1 -19732.23,E2 -19732.23} C_VEL
LIN {X 0,Y 249.142,Z 263.734,A -85,B 0,C 180,E1 -19732.765,E2 -19732.765} C_VEL
LIN {X 0,Y 251.217,Z 200.011,A -85,B 0,C 180,E1 -19734.545,E2 -19734.545} C_VEL
LIN {X 0,Y 245.601,Z 185.524,A -85,B 0,C 180,E1 -19735.706,E2 -19735.706} C_VEL
LIN {X 0,Y 238.055,Z 170.745,A -85,B 0,C 180,E1 -19737.213,E2 -19737.213} C_VEL
LIN {X 0,Y 235.249,Z 165.47,A -85,B 0,C 180,E1 -19737.796,E2 -19737.796} C_VEL
LIN {X 0,Y 234.967,Z 164.217,A -85,B 0,C 180,E1 -19737.963,E2 -19737.963} C_VEL
LIN {X 0,Y 234.958,Z 164.215,A -85,B 0,C 180,E1 -19742.573,E2 -19742.573} C_VEL
LIN {X 0,Y 234.936,Z 164.217,A -85,B 0,C 180,E1 -19746.745,E2 -19746.745} C_VEL
LIN {X 0,Y 234.938,Z 164.216,A -85,B 0,C 180,E1 -19748.942,E2 -19748.942} C_VEL
LIN {X 0,Y 234.882,Z 164.227,A -85,B 0,C 180,E1 -19753.484,E2 -19753.484} C_VEL
LIN {X 0,Y 234.882,Z 164.223,A -85,B 0,C 180,E1 -19756.512,E2 -19756.512} C_VEL
LIN {X 0,Y 234.913,Z 164.222,A -85,B 0,C 180,E1 -19761.077,E2 -19761.077} C_VEL
LIN {X 0,Y 234.924,Z 164.223,A -85,B 0,C 180,E1 -19765.361,E2 -19765.361} C_VEL
LIN {X 0,Y 234.914,Z 164.224,A -85,B 0,C 180,E1 -19769.429,E2 -19769.429} C_VEL
LIN {X 0,Y 234.985,Z 164.212,A -85,B 0,C 180,E1 -19773.793,E2 -19773.793} C_VEL
LIN {X 0,Y 234.96,Z 164.209,A -85,B 0,C 180,E1 -19778.965,E2 -19778.965} C_VEL
LIN {X 0,Y 235.047,Z 164.204,A -85,B 0,C 180,E1 -19783.091,E2 -19783.091} C_VEL
LIN {X 0,Y 235.087,Z 164.2,A -85,B 0,C 180,E1 -19787.92,E2 -19787.92} C_VEL
LIN {X 0,Y 235.301,Z 164.157,A -85,B 0,C 180,E1 -19791.411,E2 -19791.411} C_VEL
LIN {X 0,Y 235.337,Z 164.137,A -85,B 0,C 180,E1 -19793.139,E2 -19793.139} C_VEL
LIN {X 0,Y 235.564,Z 164.136,A -85,B 0,C 180,E1 -19798.29,E2 -19798.29} C_VEL
LIN {X 0,Y 235.565,Z 164.139,A -85,B 0,C 180,E1 -19801.709,E2 -19801.709} C_VEL
LIN {X 0,Y 235.337,Z 164.169,A -85,B 0,C 180,E1 -19806.86,E2 -19806.86} C_VEL
LIN {X 0,Y 235.2,Z 164.188,A -85,B 0,C 180,E1 -19810.328,E2 -19810.328} C_VEL
LIN {X 0,Y 235.065,Z 164.203,A -85,B 0,C 180,E1 -19815.61,E2 -19815.61} C_VEL
LIN {X 0,Y 234.975,Z 164.217,A -85,B 0,C 180,E1 -19819.208,E2 -19819.208} C_VEL
LIN {X 0,Y 234.958,Z 164.219,A -85,B 0,C 180,E1 -19822.145,E2 -19822.145} C_VEL
LIN {X 0,Y 234.253,Z 164.308,A -85,B 0,C 180,E1 -19823.576,E2 -19823.576} C_VEL
LIN {X 0,Y 231.407,Z 164.662,A -85,B 0,C 180,E1 -19825.911,E2 -19825.911} C_VEL
LIN {X 0,Y 229.008,Z 164.961,A -85,B 0,C 180,E1 -19827.815,E2 -19827.815} C_VEL
LIN {X 0,Y 227.975,Z 165.089,A -85,B 0,C 180,E1 -19829.292,E2 -19829.292} C_VEL
LIN {X 0,Y 227.888,Z 165.1,A -85,B 0,C 180,E1 -19829.793,E2 -19829.793} C_VEL
LIN {X 0,Y 227.87,Z 165.103,A -85,B 0,C 180,E1 -19833.722,E2 -19833.722} C_VEL
LIN {X 0,Y 227.837,Z 165.108,A -85,B 0,C 180,E1 -19838.092,E2 -19838.092} C_VEL
LIN {X 0,Y 227.805,Z 165.11,A -85,B 0,C 180,E1 -19842.744,E2 -19842.744} C_VEL
LIN {X 0,Y 227.805,Z 165.101,A -85,B 0,C 180,E1 -19847.259,E2 -19847.259} C_VEL
LIN {X 0,Y 227.903,Z 165.238,A -85,B 0,C 180,E1 -19850.679,E2 -19850.679} C_VEL
LIN {X 0,Y 230.111,Z 174.09,A -85,B 0,C 180,E1 -19854.531,E2 -19854.531} C_VEL
LIN {X 0,Y 231.133,Z 178.748,A -85,B 0,C 180,E1 -19856.452,E2 -19856.452} C_VEL
LIN {X 0,Y 238.594,Z 196.868,A -85,B 0,C 180,E1 -19858.141,E2 -19858.141} C_VEL
LIN {X 0,Y 239.752,Z 200.592,A -85,B 0,C 180,E1 -19858.422,E2 -19858.422} C_VEL
LIN {X 0,Y 243.104,Z 227.268,A -85,B 0,C 180,E1 -19859.736,E2 -19859.736} C_VEL
LIN {X 0,Y 243.841,Z 235.23,A -85,B 0,C 180,E1 -19860.086,E2 -19860.086} C_VEL
LIN {X 0,Y 241.979,Z 287.705,A -85,B 0,C 180,E1 -19861.606,E2 -19861.606} C_VEL
LIN {X 0,Y 241.016,Z 300.321,A -85,B 0,C 180,E1 -19862.25,E2 -19862.25} C_VEL
LIN {X 0,Y 239.531,Z 312.756,A -85,B 0,C 180,E1 -19863.187,E2 -19863.187} C_VEL
LIN {X 0,Y 237.724,Z 324.397,A -85,B 0,C 180,E1 -19864.384,E2 -19864.384} C_VEL
LIN {X 0,Y 235.586,Z 336.321,A -85,B 0,C 180,E1 -19866.019,E2 -19866.019} C_VEL
LIN {X 0,Y 233.349,Z 346.964,A -85,B 0,C 180,E1 -19867.887,E2 -19867.887} C_VEL
LIN {X 0,Y 231.38,Z 356.575,A -85,B 0,C 180,E1 -19870.021,E2 -19870.021} C_VEL
LIN {X 0,Y 229.862,Z 364.453,A -85,B 0,C 180,E1 -19872.199,E2 -19872.199} C_VEL
LIN {X 0,Y 228.161,Z 372.124,A -85,B 0,C 180,E1 -19874.824,E2 -19874.824} C_VEL
LIN {X 0,Y 226.873,Z 378.294,A -85,B 0,C 180,E1 -19877.478,E2 -19877.478} C_VEL
LIN {X 0,Y 226.186,Z 383.198,A -85,B 0,C 180,E1 -19880.162,E2 -19880.162} C_VEL
LIN {X 0,Y 225.821,Z 386.962,A -85,B 0,C 180,E1 -19882.851,E2 -19882.851} C_VEL
LIN {X 0,Y 225.737,Z 389.295,A -85,B 0,C 180,E1 -19885.053,E2 -19885.053} C_VEL
LIN {X 0,Y 225.824,Z 391.461,A -85,B 0,C 180,E1 -19888.218,E2 -19888.218} C_VEL
LIN {X 0,Y 225.875,Z 392.114,A -85,B 0,C 180,E1 -19890.002,E2 -19890.002} C_VEL
LIN {X 0,Y 225.802,Z 392.368,A -85,B 0,C 180,E1 -19891.785,E2 -19891.785} C_VEL
LIN {X 0,Y 225.689,Z 391.868,A -85,B 0,C 180,E1 -19894.805,E2 -19894.805} C_VEL
LIN {X 0,Y 225.766,Z 390.665,A -85,B 0,C 180,E1 -19897.154,E2 -19897.154} C_VEL
LIN {X 0,Y 226.038,Z 389.304,A -85,B 0,C 180,E1 -19898.945,E2 -19898.945} C_VEL
LIN {X 0,Y 226.757,Z 386.447,A -85,B 0,C 180,E1 -19901.624,E2 -19901.624} C_VEL
LIN {X 0,Y 227.88,Z 382.576,A -85,B 0,C 180,E1 -19904.285,E2 -19904.285} C_VEL
LIN {X 0,Y 229.654,Z 377.599,A -85,B 0,C 180,E1 -19906.903,E2 -19906.903} C_VEL
LIN {X 0,Y 231.742,Z 371.358,A -85,B 0,C 180,E1 -19909.489,E2 -19909.489} C_VEL
LIN {X 0,Y 234.115,Z 363.593,A -85,B 0,C 180,E1 -19912.041,E2 -19912.041} C_VEL
LIN {X 0,Y 237.254,Z 353.895,A -85,B 0,C 180,E1 -19914.502,E2 -19914.502} C_VEL
LIN {X 0,Y 240.238,Z 343.897,A -85,B 0,C 180,E1 -19916.497,E2 -19916.497} C_VEL
LIN {X 0,Y 243.184,Z 332.6,A -85,B 0,C 180,E1 -19918.246,E2 -19918.246} C_VEL
LIN {X 0,Y 245.657,Z 321.545,A -85,B 0,C 180,E1 -19919.572,E2 -19919.572} C_VEL
LIN {X 0,Y 247.953,Z 309.281,A -85,B 0,C 180,E1 -19920.678,E2 -19920.678} C_VEL
LIN {X 0,Y 249.71,Z 296.328,A -85,B 0,C 180,E1 -19921.497,E2 -19921.497} C_VEL
LIN {X 0,Y 250.801,Z 282.551,A -85,B 0,C 180,E1 -19922.052,E2 -19922.052} C_VEL
LIN {X 0,Y 252.632,Z 238.145,A -85,B 0,C 180,E1 -19923.279,E2 -19923.279} C_VEL
LIN {X 0,Y 249.176,Z 214.438,A -85,B 0,C 180,E1 -19924.671,E2 -19924.671} C_VEL
LIN {X 0,Y 242.142,Z 198.532,A -85,B 0,C 180,E1 -19926.505,E2 -19926.505} C_VEL
LIN {X 0,Y 236.185,Z 186.665,A -85,B 0,C 180,E1 -19928.122,E2 -19928.122} C_VEL
LIN {X 0,Y 233.376,Z 181.576,A -85,B 0,C 180,E1 -19928.907,E2 -19928.907} C_VEL
LIN {X 0,Y 231.419,Z 177.697,A -85,B 0,C 180,E1 -19929.511,E2 -19929.511} C_VEL
LIN {X 0,Y 229.289,Z 170.138,A -85,B 0,C 180,E1 -19933.284,E2 -19933.284} C_VEL
LIN {X 0,Y 227.849,Z 165.103,A -85,B 0,C 180,E1 -19936.04,E2 -19936.04} C_VEL
LIN {X 0,Y 227.832,Z 165.106,A -85,B 0,C 180,E1 -19940.462,E2 -19940.462} C_VEL
LIN {X 0,Y 227.883,Z 165.101,A -85,B 0,C 180,E1 -19944.129,E2 -19944.129} C_VEL
LIN {X 0,Y 227.859,Z 165.104,A -85,B 0,C 180,E1 -19948.376,E2 -19948.376} C_VEL
LIN {X 0,Y 227.858,Z 165.101,A -85,B 0,C 180,E1 -19952.441,E2 -19952.441} C_VEL
LIN {X 0,Y 227.893,Z 165.095,A -85,B 0,C 180,E1 -19956.365,E2 -19956.365} C_VEL
LIN {X 0,Y 227.892,Z 165.083,A -85,B 0,C 180,E1 -19960.17,E2 -19960.17} C_VEL
LIN {X 0,Y 228.001,Z 165.081,A -85,B 0,C 180,E1 -19963.894,E2 -19963.894} C_VEL
LIN {X 0,Y 228.127,Z 165.067,A -85,B 0,C 180,E1 -19969.348,E2 -19969.348} C_VEL
LIN {X 0,Y 228.295,Z 165.04,A -85,B 0,C 180,E1 -19972.927,E2 -19972.927} C_VEL
LIN {X 0,Y 228.501,Z 165.01,A -85,B 0,C 180,E1 -19978.238,E2 -19978.238} C_VEL
LIN {X 0,Y 228.534,Z 165.007,A -85,B 0,C 180,E1 -19981.762,E2 -19981.762} C_VEL
LIN {X 0,Y 228.303,Z 165.04,A -85,B 0,C 180,E1 -19987.073,E2 -19987.073} C_VEL
LIN {X 0,Y 228.146,Z 165.064,A -85,B 0,C 180,E1 -19990.651,E2 -19990.651} C_VEL
LIN {X 0,Y 228.021,Z 165.08,A -85,B 0,C 180,E1 -19996.105,E2 -19996.105} C_VEL
LIN {X 0,Y 227.929,Z 165.094,A -85,B 0,C 180,E1 -20001.717,E2 -20001.717} C_VEL
LIN {X 0,Y 227.927,Z 165.094,A -85,B 0,C 180,E1 -20006.592,E2 -20006.592} C_VEL
LIN {X 0,Y 227.878,Z 165.098,A -85,B 0,C 180,E1 -20010.281,E2 -20010.281} C_VEL
LIN {X 0,Y 227.88,Z 165.095,A -85,B 0,C 180,E1 -20013.72,E2 -20013.72} C_VEL
LIN {X 0,Y 227.847,Z 165.103,A -85,B 0,C 180,E1 -20018.091,E2 -20018.091} C_VEL
LIN {X 0,Y 227.813,Z 165.09,A -85,B 0,C 180,E1 -20022.742,E2 -20022.742} C_VEL
LIN {X 0,Y 227.848,Z 165.1,A -85,B 0,C 180,E1 -20024.831,E2 -20024.831} C_VEL
LIN {X 0,Y 228.91,Z 168.074,A -85,B 0,C 180,E1 -20025.234,E2 -20025.234} C_VEL
LIN {X 0,Y 230.833,Z 170.345,A -85,B 0,C 180,E1 -20025.762,E2 -20025.762} C_VEL
LIN {X 0,Y 233.012,Z 173.728,A -85,B 0,C 180,E1 -20026.376,E2 -20026.376} C_VEL
LIN {X 0,Y 242.238,Z 188.345,A -85,B 0,C 180,E1 -20028.81,E2 -20028.81} C_VEL
LIN {X 0,Y 247.188,Z 197.422,A -85,B 0,C 180,E1 -20030.053,E2 -20030.053} C_VEL
LIN {X 0,Y 253.711,Z 211.902,A -85,B 0,C 180,E1 -20031.674,E2 -20031.674} C_VEL
LIN {X 0,Y 251.266,Z 269.281,A -85,B 0,C 180,E1 -20033.3,E2 -20033.3} C_VEL
LIN {X 0,Y 249.982,Z 282.909,A -85,B 0,C 180,E1 -20034.001,E2 -20034.001} C_VEL
LIN {X 0,Y 248.341,Z 294.827,A -85,B 0,C 180,E1 -20034.91,E2 -20034.91} C_VEL
LIN {X 0,Y 246.358,Z 306.248,A -85,B 0,C 180,E1 -20036.105,E2 -20036.105} C_VEL
LIN {X 0,Y 243.683,Z 318.329,A -85,B 0,C 180,E1 -20037.753,E2 -20037.753} C_VEL
LIN {X 0,Y 240.943,Z 328.638,A -85,B 0,C 180,E1 -20039.547,E2 -20039.547} C_VEL
LIN {X 0,Y 238.527,Z 337.042,A -85,B 0,C 180,E1 -20041.392,E2 -20041.392} C_VEL
LIN {X 0,Y 235.744,Z 346.121,A -85,B 0,C 180,E1 -20043.912,E2 -20043.912} C_VEL
LIN {X 0,Y 233.161,Z 353.415,A -85,B 0,C 180,E1 -20046.459,E2 -20046.459} C_VEL
LIN {X 0,Y 231.349,Z 358.334,A -85,B 0,C 180,E1 -20048.619,E2 -20048.619} C_VEL
LIN {X 0,Y 229.488,Z 363.234,A -85,B 0,C 180,E1 -20051.334,E2 -20051.334} C_VEL
LIN {X 0,Y 228.087,Z 366.727,A -85,B 0,C 180,E1 -20053.899,E2 -20053.899} C_VEL
LIN {X 0,Y 227.365,Z 368.595,A -85,B 0,C 180,E1 -20055.682,E2 -20055.682} C_VEL
LIN {X 0,Y 226.753,Z 370.007,A -85,B 0,C 180,E1 -20057.468,E2 -20057.468} C_VEL
LIN {X 0,Y 226.096,Z 371.6,A -85,B 0,C 180,E1 -20061.057,E2 -20061.057} C_VEL
LIN {X 0,Y 225.955,Z 371.67,A -85,B 0,C 180,E1 -20064.456,E2 -20064.456} C_VEL
LIN {X 0,Y 225.893,Z 371.028,A -85,B 0,C 180,E1 -20066.431,E2 -20066.431} C_VEL
LIN {X 0,Y 225.932,Z 370.056,A -85,B 0,C 180,E1 -20068.216,E2 -20068.216} C_VEL
LIN {X 0,Y 226.022,Z 368.7,A -85,B 0,C 180,E1 -20069.998,E2 -20069.998} C_VEL
LIN {X 0,Y 226.524,Z 365.831,A -85,B 0,C 180,E1 -20072.666,E2 -20072.666} C_VEL
LIN {X 0,Y 227.247,Z 361.952,A -85,B 0,C 180,E1 -20075.322,E2 -20075.322} C_VEL
LIN {X 0,Y 228.396,Z 356.948,A -85,B 0,C 180,E1 -20077.958,E2 -20077.958} C_VEL
LIN {X 0,Y 229.701,Z 350.673,A -85,B 0,C 180,E1 -20080.576,E2 -20080.576} C_VEL
LIN {X 0,Y 231.667,Z 342.795,A -85,B 0,C 180,E1 -20083.15,E2 -20083.15} C_VEL
LIN {X 0,Y 233.538,Z 334.363,A -85,B 0,C 180,E1 -20085.372,E2 -20085.372} C_VEL
LIN {X 0,Y 235.669,Z 323.945,A -85,B 0,C 180,E1 -20087.572,E2 -20087.572} C_VEL
LIN {X 0,Y 237.702,Z 312.66,A -85,B 0,C 180,E1 -20089.426,E2 -20089.426} C_VEL
LIN {X 0,Y 239.484,Z 301.593,A -85,B 0,C 180,E1 -20090.842,E2 -20090.842} C_VEL
LIN {X 0,Y 240.925,Z 289.284,A -85,B 0,C 180,E1 -20092.058,E2 -20092.058} C_VEL
LIN {X 0,Y 242.082,Z 276.136,A -85,B 0,C 180,E1 -20092.959,E2 -20092.959} C_VEL
LIN {X 0,Y 242.81,Z 263.391,A -85,B 0,C 180,E1 -20093.507,E2 -20093.507} C_VEL
LIN {X 0,Y 244.941,Z 201.643,A -85,B 0,C 180,E1 -20095.263,E2 -20095.263} C_VEL
LIN {X 0,Y 239.429,Z 187.839,A -85,B 0,C 180,E1 -20096.442,E2 -20096.442} C_VEL
LIN {X 0,Y 232.547,Z 174.374,A -85,B 0,C 180,E1 -20097.88,E2 -20097.88} C_VEL
LIN {X 0,Y 228.909,Z 167.921,A -85,B 0,C 180,E1 -20098.66,E2 -20098.66} C_VEL
LIN {X 0,Y 227.919,Z 165.092,A -85,B 0,C 180,E1 -20098.962,E2 -20098.962} C_VEL
LIN {X 0,Y 227.888,Z 165.097,A -85,B 0,C 180,E1 -20103.716,E2 -20103.716} C_VEL
LIN {X 0,Y 227.846,Z 165.101,A -85,B 0,C 180,E1 -20108.088,E2 -20108.088} C_VEL
LIN {X 0,Y 227.806,Z 165.107,A -85,B 0,C 180,E1 -20112.74,E2 -20112.74} C_VEL
LIN {X 0,Y 227.806,Z 165.104,A -85,B 0,C 180,E1 -20117.256,E2 -20117.256} C_VEL
LIN {X 0,Y 227.838,Z 165.1,A -85,B 0,C 180,E1 -20121.907,E2 -20121.907} C_VEL
LIN {X 0,Y 227.873,Z 165.095,A -85,B 0,C 180,E1 -20126.376,E2 -20126.376} C_VEL
LIN {X 0,Y 227.894,Z 165.097,A -85,B 0,C 180,E1 -20130.434,E2 -20130.434} C_VEL
LIN {X 0,Y 227.916,Z 165.093,A -85,B 0,C 180,E1 -20134.424,E2 -20134.424} C_VEL
LIN {X 0,Y 227.93,Z 165.084,A -85,B 0,C 180,E1 -20138.284,E2 -20138.284} C_VEL
LIN {X 0,Y 227.982,Z 165.085,A -85,B 0,C 180,E1 -20142.861,E2 -20142.861} C_VEL
LIN {X 0,Y 228.045,Z 165.079,A -85,B 0,C 180,E1 -20147.541,E2 -20147.541} C_VEL
LIN {X 0,Y 228.243,Z 165.038,A -85,B 0,C 180,E1 -20151.143,E2 -20151.143} C_VEL
LIN {X 0,Y 228.29,Z 165.015,A -85,B 0,C 180,E1 -20152.926,E2 -20152.926} C_VEL
LIN {X 0,Y 228.523,Z 165.013,A -85,B 0,C 180,E1 -20158.237,E2 -20158.237} C_VEL
LIN {X 0,Y 228.524,Z 165.016,A -85,B 0,C 180,E1 -20161.762,E2 -20161.762} C_VEL
LIN {X 0,Y 228.289,Z 165.046,A -85,B 0,C 180,E1 -20167.073,E2 -20167.073} C_VEL
LIN {X 0,Y 228.131,Z 165.07,A -85,B 0,C 180,E1 -20170.652,E2 -20170.652} C_VEL
LIN {X 0,Y 228.024,Z 165.083,A -85,B 0,C 180,E1 -20174.275,E2 -20174.275} C_VEL
LIN {X 0,Y 227.942,Z 165.093,A -85,B 0,C 180,E1 -20177.958,E2 -20177.958} C_VEL
LIN {X 0,Y 227.906,Z 165.099,A -85,B 0,C 180,E1 -20182.32,E2 -20182.32} C_VEL
LIN {X 0,Y 227.932,Z 165.099,A -85,B 0,C 180,E1 -20186.602,E2 -20186.602} C_VEL
LIN {X 0,Y 227.888,Z 165.1,A -85,B 0,C 180,E1 -20189.793,E2 -20189.793} C_VEL
LIN {X 0,Y 227.215,Z 165.188,A -85,B 0,C 180,E1 -20191.268,E2 -20191.268} C_VEL
LIN {X 0,Y 224.38,Z 165.547,A -85,B 0,C 180,E1 -20193.677,E2 -20193.677} C_VEL
LIN {X 0,Y 221.127,Z 165.945,A -85,B 0,C 180,E1 -20196.652,E2 -20196.652} C_VEL
LIN {X 0,Y 220.777,Z 165.983,A -85,B 0,C 180,E1 -20197.683,E2 -20197.683} C_VEL
LIN {X 0,Y 220.763,Z 165.988,A -85,B 0,C 180,E1 -20201.954,E2 -20201.954} C_VEL
LIN {X 0,Y 220.768,Z 165.985,A -85,B 0,C 180,E1 -20205.548,E2 -20205.548} C_VEL
LIN {X 0,Y 220.795,Z 166.107,A -85,B 0,C 180,E1 -20209.812,E2 -20209.812} C_VEL
LIN {X 0,Y 223.046,Z 174.573,A -85,B 0,C 180,E1 -20213.684,E2 -20213.684} C_VEL
LIN {X 0,Y 223.912,Z 178.486,A -85,B 0,C 180,E1 -20215.331,E2 -20215.331} C_VEL
LIN {X 0,Y 231.855,Z 197.289,A -85,B 0,C 180,E1 -20217.217,E2 -20217.217} C_VEL
LIN {X 0,Y 233.753,Z 203.047,A -85,B 0,C 180,E1 -20217.688,E2 -20217.688} C_VEL
LIN {X 0,Y 236.982,Z 229.678,A -85,B 0,C 180,E1 -20219.036,E2 -20219.036} C_VEL
LIN {X 0,Y 237.505,Z 236.55,A -85,B 0,C 180,E1 -20219.336,E2 -20219.336} C_VEL
LIN {X 0,Y 235.598,Z 287.868,A -85,B 0,C 180,E1 -20220.866,E2 -20220.866} C_VEL
LIN {X 0,Y 234.568,Z 300.578,A -85,B 0,C 180,E1 -20221.54,E2 -20221.54} C_VEL
LIN {X 0,Y 233.043,Z 312.864,A -85,B 0,C 180,E1 -20222.5,E2 -20222.5} C_VEL
LIN {X 0,Y 231.03,Z 325.23,A -85,B 0,C 180,E1 -20223.828,E2 -20223.828} C_VEL
LIN {X 0,Y 228.83,Z 336.895,A -85,B 0,C 180,E1 -20225.507,E2 -20225.507} C_VEL
LIN {X 0,Y 226.511,Z 347.383,A -85,B 0,C 180,E1 -20227.423,E2 -20227.423} C_VEL
LIN {X 0,Y 224.661,Z 355.973,A -85,B 0,C 180,E1 -20229.397,E2 -20229.397} C_VEL
LIN {X 0,Y 223.055,Z 363.905,A -85,B 0,C 180,E1 -20231.636,E2 -20231.636} C_VEL
LIN {X 0,Y 221.283,Z 371.625,A -85,B 0,C 180,E1 -20234.34,E2 -20234.34} C_VEL
LIN {X 0,Y 219.9,Z 377.827,A -85,B 0,C 180,E1 -20237.074,E2 -20237.074} C_VEL
LIN {X 0,Y 219.139,Z 382.76,A -85,B 0,C 180,E1 -20239.842,E2 -20239.842} C_VEL
LIN {X 0,Y 218.749,Z 386.554,A -85,B 0,C 180,E1 -20242.618,E2 -20242.618} C_VEL
LIN {X 0,Y 218.643,Z 389.139,A -85,B 0,C 180,E1 -20245.175,E2 -20245.175} C_VEL
LIN {X 0,Y 218.732,Z 391.106,A -85,B 0,C 180,E1 -20248.16,E2 -20248.16} C_VEL
LIN {X 0,Y 218.806,Z 391.773,A -85,B 0,C 180,E1 -20250.002,E2 -20250.002} C_VEL
LIN {X 0,Y 218.708,Z 392.038,A -85,B 0,C 180,E1 -20251.843,E2 -20251.843} C_VEL
LIN {X 0,Y 218.589,Z 391.646,A -85,B 0,C 180,E1 -20254.655,E2 -20254.655} C_VEL
LIN {X 0,Y 218.688,Z 390.383,A -85,B 0,C 180,E1 -20257.387,E2 -20257.387} C_VEL
LIN {X 0,Y 219.003,Z 389.035,A -85,B 0,C 180,E1 -20259.235,E2 -20259.235} C_VEL
LIN {X 0,Y 219.765,Z 386.203,A -85,B 0,C 180,E1 -20261.999,E2 -20261.999} C_VEL
LIN {X 0,Y 220.993,Z 382.361,A -85,B 0,C 180,E1 -20264.74,E2 -20264.74} C_VEL
LIN {X 0,Y 222.83,Z 377.414,A -85,B 0,C 180,E1 -20267.437,E2 -20267.437} C_VEL
LIN {X 0,Y 225.011,Z 371.206,A -85,B 0,C 180,E1 -20270.096,E2 -20270.096} C_VEL
LIN {X 0,Y 227.538,Z 363.498,A -85,B 0,C 180,E1 -20272.713,E2 -20272.713} C_VEL
LIN {X 0,Y 230.81,Z 353.849,A -85,B 0,C 180,E1 -20275.234,E2 -20275.234} C_VEL
LIN {X 0,Y 233.899,Z 343.912,A -85,B 0,C 180,E1 -20277.274,E2 -20277.274} C_VEL
LIN {X 0,Y 236.961,Z 332.724,A -85,B 0,C 180,E1 -20279.057,E2 -20279.057} C_VEL
LIN {X 0,Y 239.527,Z 321.777,A -85,B 0,C 180,E1 -20280.408,E2 -20280.408} C_VEL
LIN {X 0,Y 241.886,Z 309.672,A -85,B 0,C 180,E1 -20281.534,E2 -20281.534} C_VEL
LIN {X 0,Y 243.728,Z 297.153,A -85,B 0,C 180,E1 -20282.363,E2 -20282.363} C_VEL
LIN {X 0,Y 244.864,Z 284.113,A -85,B 0,C 180,E1 -20282.926,E2 -20282.926} C_VEL
LIN {X 0,Y 246.841,Z 239.269,A -85,B 0,C 180,E1 -20284.193,E2 -20284.193} C_VEL
LIN {X 0,Y 243.613,Z 216.985,A -85,B 0,C 180,E1 -20285.556,E2 -20285.556} C_VEL
LIN {X 0,Y 236.747,Z 201.34,A -85,B 0,C 180,E1 -20287.441,E2 -20287.441} C_VEL
LIN {X 0,Y 229.434,Z 186.933,A -85,B 0,C 180,E1 -20289.545,E2 -20289.545} C_VEL
LIN {X 0,Y 226.335,Z 181.554,A -85,B 0,C 180,E1 -20290.469,E2 -20290.469} C_VEL
LIN {X 0,Y 224.054,Z 177.272,A -85,B 0,C 180,E1 -20291.203,E2 -20291.203} C_VEL
LIN {X 0,Y 221.884,Z 169.895,A -85,B 0,C 180,E1 -20295.155,E2 -20295.155} C_VEL
LIN {X 0,Y 220.754,Z 165.986,A -85,B 0,C 180,E1 -20297.453,E2 -20297.453} C_VEL
LIN {X 0,Y 220.786,Z 165.984,A -85,B 0,C 180,E1 -20300.459,E2 -20300.459} C_VEL
LIN {X 0,Y 220.828,Z 165.978,A -85,B 0,C 180,E1 -20302.794,E2 -20302.794} C_VEL
LIN {X 0,Y 220.815,Z 165.979,A -85,B 0,C 180,E1 -20307.244,E2 -20307.244} C_VEL
LIN {X 0,Y 220.807,Z 165.978,A -85,B 0,C 180,E1 -20311.482,E2 -20311.482} C_VEL
LIN {X 0,Y 220.848,Z 165.975,A -85,B 0,C 180,E1 -20315.563,E2 -20315.563} C_VEL
LIN {X 0,Y 220.851,Z 165.963,A -85,B 0,C 180,E1 -20319.51,E2 -20319.51} C_VEL
LIN {X 0,Y 220.968,Z 165.959,A -85,B 0,C 180,E1 -20323.367,E2 -20323.367} C_VEL
LIN {X 0,Y 221.052,Z 165.949,A -85,B 0,C 180,E1 -20329.003,E2 -20329.003} C_VEL
LIN {X 0,Y 221.232,Z 165.917,A -85,B 0,C 180,E1 -20332.7,E2 -20332.7} C_VEL
LIN {X 0,Y 221.438,Z 165.888,A -85,B 0,C 180,E1 -20338.181,E2 -20338.181} C_VEL
LIN {X 0,Y 221.544,Z 165.89,A -85,B 0,C 180,E1 -20340,E2 -20340} C_VEL
LIN {X 0,Y 221.467,Z 165.886,A -85,B 0,C 180,E1 -20341.819,E2 -20341.819} C_VEL
LIN {X 0,Y 221.241,Z 165.917,A -85,B 0,C 180,E1 -20347.3,E2 -20347.3} C_VEL
LIN {X 0,Y 221.066,Z 165.947,A -85,B 0,C 180,E1 -20350.997,E2 -20350.997} C_VEL
LIN {X 0,Y 220.98,Z 165.958,A -85,B 0,C 180,E1 -20356.633,E2 -20356.633} C_VEL
LIN {X 0,Y 220.857,Z 165.964,A -85,B 0,C 180,E1 -20360.49,E2 -20360.49} C_VEL
LIN {X 0,Y 220.849,Z 165.963,A -85,B 0,C 180,E1 -20364.438,E2 -20364.438} C_VEL
LIN {X 0,Y 220.808,Z 165.971,A -85,B 0,C 180,E1 -20368.518,E2 -20368.518} C_VEL
LIN {X 0,Y 220.816,Z 165.971,A -85,B 0,C 180,E1 -20372.757,E2 -20372.757} C_VEL
LIN {X 0,Y 220.814,Z 165.974,A -85,B 0,C 180,E1 -20377.278,E2 -20377.278} C_VEL
LIN {X 0,Y 220.77,Z 165.959,A -85,B 0,C 180,E1 -20381.953,E2 -20381.953} C_VEL
LIN {X 0,Y 220.782,Z 166.131,A -85,B 0,C 180,E1 -20383.19,E2 -20383.19} C_VEL
LIN {X 0,Y 221.701,Z 168.73,A -85,B 0,C 180,E1 -20383.538,E2 -20383.538} C_VEL
LIN {X 0,Y 223.826,Z 171.189,A -85,B 0,C 180,E1 -20384.169,E2 -20384.169} C_VEL
LIN {X 0,Y 226.022,Z 174.634,A -85,B 0,C 180,E1 -20384.841,E2 -20384.841} C_VEL
LIN {X 0,Y 232.41,Z 184.354,A -85,B 0,C 180,E1 -20386.673,E2 -20386.673} C_VEL
LIN {X 0,Y 239.624,Z 196.312,A -85,B 0,C 180,E1 -20388.607,E2 -20388.607} C_VEL
LIN {X 0,Y 244.914,Z 207.049,A -85,B 0,C 180,E1 -20389.993,E2 -20389.993} C_VEL
LIN {X 0,Y 247.897,Z 213.987,A -85,B 0,C 180,E1 -20390.769,E2 -20390.769} C_VEL
LIN {X 0,Y 245.434,Z 269.439,A -85,B 0,C 180,E1 -20392.368,E2 -20392.368} C_VEL
LIN {X 0,Y 244.142,Z 282.823,A -85,B 0,C 180,E1 -20393.063,E2 -20393.063} C_VEL
LIN {X 0,Y 242.336,Z 295.403,A -85,B 0,C 180,E1 -20394.035,E2 -20394.035} C_VEL
LIN {X 0,Y 240.294,Z 306.709,A -85,B 0,C 180,E1 -20395.248,E2 -20395.248} C_VEL
LIN {X 0,Y 237.663,Z 318.156,A -85,B 0,C 180,E1 -20396.832,E2 -20396.832} C_VEL
LIN {X 0,Y 234.814,Z 328.558,A -85,B 0,C 180,E1 -20398.664,E2 -20398.664} C_VEL
LIN {X 0,Y 232.249,Z 337.037,A -85,B 0,C 180,E1 -20400.544,E2 -20400.544} C_VEL
LIN {X 0,Y 229.31,Z 346.185,A -85,B 0,C 180,E1 -20403.122,E2 -20403.122} C_VEL
LIN {X 0,Y 226.624,Z 353.524,A -85,B 0,C 180,E1 -20405.737,E2 -20405.737} C_VEL
LIN {X 0,Y 224.002,Z 360.228,A -85,B 0,C 180,E1 -20408.849,E2 -20408.849} C_VEL
LIN {X 0,Y 222.181,Z 364.707,A -85,B 0,C 180,E1 -20411.616,E2 -20411.616} C_VEL
LIN {X 0,Y 221.206,Z 366.949,A -85,B 0,C 180,E1 -20413.383,E2 -20413.383} C_VEL
LIN {X 0,Y 220.419,Z 368.835,A -85,B 0,C 180,E1 -20415.22,E2 -20415.22} C_VEL
LIN {X 0,Y 219.767,Z 370.279,A -85,B 0,C 180,E1 -20417.063,E2 -20417.063} C_VEL
LIN {X 0,Y 219.033,Z 371.903,A -85,B 0,C 180,E1 -20420.766,E2 -20420.766} C_VEL
LIN {X 0,Y 218.926,Z 372.138,A -85,B 0,C 180,E1 -20422.621,E2 -20422.621} C_VEL
LIN {X 0,Y 218.845,Z 371.937,A -85,B 0,C 180,E1 -20424.59,E2 -20424.59} C_VEL
LIN {X 0,Y 218.861,Z 370.433,A -85,B 0,C 180,E1 -20428.158,E2 -20428.158} C_VEL
LIN {X 0,Y 218.946,Z 369.093,A -85,B 0,C 180,E1 -20429.998,E2 -20429.998} C_VEL
LIN {X 0,Y 219.445,Z 366.257,A -85,B 0,C 180,E1 -20432.752,E2 -20432.752} C_VEL
LIN {X 0,Y 220.195,Z 362.413,A -85,B 0,C 180,E1 -20435.493,E2 -20435.493} C_VEL
LIN {X 0,Y 221.381,Z 357.446,A -85,B 0,C 180,E1 -20438.211,E2 -20438.211} C_VEL
LIN {X 0,Y 222.76,Z 351.223,A -85,B 0,C 180,E1 -20440.91,E2 -20440.91} C_VEL
LIN {X 0,Y 224.799,Z 343.404,A -85,B 0,C 180,E1 -20443.559,E2 -20443.559} C_VEL
LIN {X 0,Y 226.65,Z 335.466,A -85,B 0,C 180,E1 -20445.737,E2 -20445.737} C_VEL
LIN {X 0,Y 228.717,Z 325.755,A -85,B 0,C 180,E1 -20447.893,E2 -20447.893} C_VEL
LIN {X 0,Y 230.839,Z 314.939,A -85,B 0,C 180,E1 -20449.796,E2 -20449.796} C_VEL
LIN {X 0,Y 232.898,Z 302.595,A -85,B 0,C 180,E1 -20451.46,E2 -20451.46} C_VEL
LIN {X 0,Y 234.423,Z 290.508,A -85,B 0,C 180,E1 -20452.703,E2 -20452.703} C_VEL
LIN {X 0,Y 235.621,Z 277.861,A -85,B 0,C 180,E1 -20453.627,E2 -20453.627} C_VEL
LIN {X 0,Y 236.448,Z 264.524,A -85,B 0,C 180,E1 -20454.237,E2 -20454.237} C_VEL
LIN {X 0,Y 238.676,Z 203.379,A -85,B 0,C 180,E1 -20456.018,E2 -20456.018} C_VEL
LIN {X 0,Y 233.711,Z 191.004,A -85,B 0,C 180,E1 -20457.127,E2 -20457.127} C_VEL
LIN {X 0,Y 226.191,Z 176.263,A -85,B 0,C 180,E1 -20458.78,E2 -20458.78} C_VEL
LIN {X 0,Y 222.203,Z 169.312,A -85,B 0,C 180,E1 -20459.681,E2 -20459.681} C_VEL
LIN {X 0,Y 220.968,Z 166.508,A -85,B 0,C 180,E1 -20459.994,E2 -20459.994} C_VEL
LIN {X 0,Y 220.871,Z 165.971,A -85,B 0,C 180,E1 -20460.078,E2 -20460.078} C_VEL
LIN {X 0,Y 220.812,Z 165.977,A -85,B 0,C 180,E1 -20464.95,E2 -20464.95} C_VEL
LIN {X 0,Y 220.835,Z 165.974,A -85,B 0,C 180,E1 -20467.286,E2 -20467.286} C_VEL
LIN {X 0,Y 220.766,Z 165.985,A -85,B 0,C 180,E1 -20471.951,E2 -20471.951} C_VEL
LIN {X 0,Y 220.769,Z 165.986,A -85,B 0,C 180,E1 -20475.544,E2 -20475.544} C_VEL
LIN {X 0,Y 220.801,Z 165.98,A -85,B 0,C 180,E1 -20480.461,E2 -20480.461} C_VEL
LIN {X 0,Y 220.795,Z 165.982,A -85,B 0,C 180,E1 -20485.044,E2 -20485.044} C_VEL
LIN {X 0,Y 220.827,Z 165.978,A -85,B 0,C 180,E1 -20489.388,E2 -20489.388} C_VEL
LIN {X 0,Y 220.885,Z 165.966,A -85,B 0,C 180,E1 -20493.548,E2 -20493.548} C_VEL
LIN {X 0,Y 220.855,Z 165.968,A -85,B 0,C 180,E1 -20497.551,E2 -20497.551} C_VEL
LIN {X 0,Y 220.92,Z 165.964,A -85,B 0,C 180,E1 -20502.617,E2 -20502.617} C_VEL
LIN {X 0,Y 220.983,Z 165.958,A -85,B 0,C 180,E1 -20507.137,E2 -20507.137} C_VEL
LIN {X 0,Y 221.184,Z 165.919,A -85,B 0,C 180,E1 -20510.858,E2 -20510.858} C_VEL
LIN {X 0,Y 221.228,Z 165.895,A -85,B 0,C 180,E1 -20512.699,E2 -20512.699} C_VEL
LIN {X 0,Y 221.456,Z 165.893,A -85,B 0,C 180,E1 -20518.181,E2 -20518.181} C_VEL
LIN {X 0,Y 221.457,Z 165.896,A -85,B 0,C 180,E1 -20521.818,E2 -20521.818} C_VEL
LIN {X 0,Y 221.226,Z 165.925,A -85,B 0,C 180,E1 -20527.3,E2 -20527.3} C_VEL
LIN {X 0,Y 221.052,Z 165.948,A -85,B 0,C 180,E1 -20530.997,E2 -20530.997} C_VEL
LIN {X 0,Y 220.969,Z 165.959,A -85,B 0,C 180,E1 -20536.633,E2 -20536.633} C_VEL
LIN {X 0,Y 220.864,Z 165.974,A -85,B 0,C 180,E1 -20540.489,E2 -20540.489} C_VEL
LIN {X 0,Y 220.853,Z 165.976,A -85,B 0,C 180,E1 -20544.437,E2 -20544.437} C_VEL
LIN {X 0,Y 220.816,Z 165.981,A -85,B 0,C 180,E1 -20548.516,E2 -20548.516} C_VEL
LIN {X 0,Y 220.809,Z 165.984,A -85,B 0,C 180,E1 -20552.757,E2 -20552.757} C_VEL
LIN {X 0,Y 220.803,Z 165.983,A -85,B 0,C 180,E1 -20557.28,E2 -20557.28} C_VEL
LIN {X 0,Y 220.777,Z 165.983,A -85,B 0,C 180,E1 -20557.683,E2 -20557.683} C_VEL
LIN {X 0,Y 220.047,Z 166.078,A -85,B 0,C 180,E1 -20559.203,E2 -20559.203} C_VEL
LIN {X 0,Y 217.127,Z 166.44,A -85,B 0,C 180,E1 -20561.683,E2 -20561.683} C_VEL
LIN {X 0,Y 214.708,Z 166.741,A -85,B 0,C 180,E1 -20563.709,E2 -20563.709} C_VEL
LIN {X 0,Y 213.721,Z 166.863,A -85,B 0,C 180,E1 -20565.284,E2 -20565.284} C_VEL
LIN {X 0,Y 213.665,Z 166.865,A -85,B 0,C 180,E1 -20565.817,E2 -20565.817} C_VEL
LIN {X 0,Y 213.713,Z 166.964,A -85,B 0,C 180,E1 -20568.878,E2 -20568.878} C_VEL
LIN {X 0,Y 215.944,Z 175.326,A -85,B 0,C 180,E1 -20572.877,E2 -20572.877} C_VEL
LIN {X 0,Y 216.648,Z 178.186,A -85,B 0,C 180,E1 -20574.107,E2 -20574.107} C_VEL
LIN {X 0,Y 224.932,Z 197.153,A -85,B 0,C 180,E1 -20576.18,E2 -20576.18} C_VEL
LIN {X 0,Y 227.668,Z 204.478,A -85,B 0,C 180,E1 -20576.86,E2 -20576.86} C_VEL
LIN {X 0,Y 230.793,Z 230.773,A -85,B 0,C 180,E1 -20578.24,E2 -20578.24} C_VEL
LIN {X 0,Y 231.233,Z 237.34,A -85,B 0,C 180,E1 -20578.53,E2 -20578.53} C_VEL
LIN {X 0,Y 229.282,Z 287.839,A -85,B 0,C 180,E1 -20580.078,E2 -20580.078} C_VEL
LIN {X 0,Y 228.16,Z 300.819,A -85,B 0,C 180,E1 -20580.791,E2 -20580.791} C_VEL
LIN {X 0,Y 226.573,Z 312.958,A -85,B 0,C 180,E1 -20581.771,E2 -20581.771} C_VEL
LIN {X 0,Y 224.647,Z 324.396,A -85,B 0,C 180,E1 -20583.026,E2 -20583.026} C_VEL
LIN {X 0,Y 222.337,Z 336.16,A -85,B 0,C 180,E1 -20584.742,E2 -20584.742} C_VEL
LIN {X 0,Y 219.977,Z 346.725,A -85,B 0,C 180,E1 -20586.713,E2 -20586.713} C_VEL
LIN {X 0,Y 217.978,Z 355.366,A -85,B 0,C 180,E1 -20588.735,E2 -20588.735} C_VEL
LIN {X 0,Y 216.251,Z 363.348,A -85,B 0,C 180,E1 -20591.037,E2 -20591.037} C_VEL
LIN {X 0,Y 214.414,Z 371.125,A -85,B 0,C 180,E1 -20593.825,E2 -20593.825} C_VEL
LIN {X 0,Y 212.936,Z 377.36,A -85,B 0,C 180,E1 -20596.644,E2 -20596.644} C_VEL
LIN {X 0,Y 212.098,Z 382.323,A -85,B 0,C 180,E1 -20599.501,E2 -20599.501} C_VEL
LIN {X 0,Y 211.669,Z 386.146,A -85,B 0,C 180,E1 -20602.37,E2 -20602.37} C_VEL
LIN {X 0,Y 211.544,Z 388.999,A -85,B 0,C 180,E1 -20605.326,E2 -20605.326} C_VEL
LIN {X 0,Y 211.641,Z 390.752,A -85,B 0,C 180,E1 -20608.099,E2 -20608.099} C_VEL
LIN {X 0,Y 211.738,Z 391.432,A -85,B 0,C 180,E1 -20610.002,E2 -20610.002} C_VEL
LIN {X 0,Y 211.617,Z 391.708,A -85,B 0,C 180,E1 -20611.905,E2 -20611.905} C_VEL
LIN {X 0,Y 211.514,Z 391.404,A -85,B 0,C 180,E1 -20614.574,E2 -20614.574} C_VEL
LIN {X 0,Y 211.628,Z 390.102,A -85,B 0,C 180,E1 -20617.635,E2 -20617.635} C_VEL
LIN {X 0,Y 211.983,Z 388.766,A -85,B 0,C 180,E1 -20619.543,E2 -20619.543} C_VEL
LIN {X 0,Y 212.79,Z 385.961,A -85,B 0,C 180,E1 -20622.398,E2 -20622.398} C_VEL
LIN {X 0,Y 214.12,Z 382.148,A -85,B 0,C 180,E1 -20625.225,E2 -20625.225} C_VEL
LIN {X 0,Y 216.016,Z 377.23,A -85,B 0,C 180,E1 -20628.005,E2 -20628.005} C_VEL
LIN {X 0,Y 218.317,Z 371.056,A -85,B 0,C 180,E1 -20630.74,E2 -20630.74} C_VEL
LIN {X 0,Y 220.979,Z 363.4,A -85,B 0,C 180,E1 -20633.427,E2 -20633.427} C_VEL
LIN {X 0,Y 223.791,Z 355.587,A -85,B 0,C 180,E1 -20635.584,E2 -20635.584} C_VEL
LIN {X 0,Y 227.256,Z 344.994,A -85,B 0,C 180,E1 -20637.89,E2 -20637.89} C_VEL
LIN {X 0,Y 230.428,Z 334.229,A -85,B 0,C 180,E1 -20639.712,E2 -20639.712} C_VEL
LIN {X 0,Y 233.099,Z 323.766,A -85,B 0,C 180,E1 -20641.087,E2 -20641.087} C_VEL
LIN {X 0,Y 235.709,Z 311.185,A -85,B 0,C 180,E1 -20642.334,E2 -20642.334} C_VEL
LIN {X 0,Y 237.791,Z 297.897,A -85,B 0,C 180,E1 -20643.274,E2 -20643.274} C_VEL
LIN {X 0,Y 238.978,Z 285.676,A -85,B 0,C 180,E1 -20643.845,E2 -20643.845} C_VEL
LIN {X 0,Y 241.103,Z 240.199,A -85,B 0,C 180,E1 -20645.16,E2 -20645.16} C_VEL
LIN {X 0,Y 238.211,Z 219.739,A -85,B 0,C 180,E1 -20646.455,E2 -20646.455} C_VEL
LIN {X 0,Y 231.334,Z 204.071,A -85,B 0,C 180,E1 -20648.441,E2 -20648.441} C_VEL
LIN {X 0,Y 224.852,Z 191.216,A -85,B 0,C 180,E1 -20650.405,E2 -20650.405} C_VEL
LIN {X 0,Y 219.061,Z 181.178,A -85,B 0,C 180,E1 -20652.25,E2 -20652.25} C_VEL
LIN {X 0,Y 216.625,Z 176.739,A -85,B 0,C 180,E1 -20653.124,E2 -20653.124} C_VEL
LIN {X 0,Y 214.249,Z 168.781,A -85,B 0,C 180,E1 -20657.743,E2 -20657.743} C_VEL
LIN {X 0,Y 213.72,Z 166.862,A -85,B 0,C 180,E1 -20659.013,E2 -20659.013} C_VEL
LIN {X 0,Y 213.747,Z 166.862,A -85,B 0,C 180,E1 -20663.712,E2 -20663.712} C_VEL
LIN {X 0,Y 213.762,Z 166.86,A -85,B 0,C 180,E1 -20668.262,E2 -20668.262} C_VEL
LIN {X 0,Y 213.792,Z 166.854,A -85,B 0,C 180,E1 -20672.599,E2 -20672.599} C_VEL
LIN {X 0,Y 213.803,Z 166.85,A -85,B 0,C 180,E1 -20676.987,E2 -20676.987} C_VEL
LIN {X 0,Y 213.881,Z 166.843,A -85,B 0,C 180,E1 -20682.799,E2 -20682.799} C_VEL
LIN {X 0,Y 213.912,Z 166.825,A -85,B 0,C 180,E1 -20686.704,E2 -20686.704} C_VEL
LIN {X 0,Y 214.126,Z 166.799,A -85,B 0,C 180,E1 -20690.555,E2 -20690.555} C_VEL
LIN {X 0,Y 214.068,Z 166.821,A -85,B 0,C 180,E1 -20694.348,E2 -20694.348} C_VEL
LIN {X 0,Y 214.378,Z 166.767,A -85,B 0,C 180,E1 -20698.122,E2 -20698.122} C_VEL
LIN {X 0,Y 214.512,Z 166.766,A -85,B 0,C 180,E1 -20700,E2 -20700} C_VEL
LIN {X 0,Y 214.404,Z 166.765,A -85,B 0,C 180,E1 -20701.879,E2 -20701.879} C_VEL
LIN {X 0,Y 214.183,Z 166.793,A -85,B 0,C 180,E1 -20707.542,E2 -20707.542} C_VEL
LIN {X 0,Y 213.995,Z 166.83,A -85,B 0,C 180,E1 -20711.365,E2 -20711.365} C_VEL
LIN {X 0,Y 213.887,Z 166.83,A -85,B 0,C 180,E1 -20715.241,E2 -20715.241} C_VEL
LIN {X 0,Y 213.8,Z 166.84,A -85,B 0,C 180,E1 -20719.191,E2 -20719.191} C_VEL
LIN {X 0,Y 213.798,Z 166.846,A -85,B 0,C 180,E1 -20723.233,E2 -20723.233} C_VEL
LIN {X 0,Y 213.791,Z 166.851,A -85,B 0,C 180,E1 -20727.428,E2 -20727.428} C_VEL
LIN {X 0,Y 213.763,Z 166.854,A -85,B 0,C 180,E1 -20731.739,E2 -20731.739} C_VEL
LIN {X 0,Y 213.748,Z 166.851,A -85,B 0,C 180,E1 -20736.288,E2 -20736.288} C_VEL
LIN {X 0,Y 213.714,Z 166.834,A -85,B 0,C 180,E1 -20741.321,E2 -20741.321} C_VEL
LIN {X 0,Y 214.595,Z 169.436,A -85,B 0,C 180,E1 -20741.701,E2 -20741.701} C_VEL
LIN {X 0,Y 216.949,Z 172.3,A -85,B 0,C 180,E1 -20742.472,E2 -20742.472} C_VEL
LIN {X 0,Y 219.207,Z 175.734,A -85,B 0,C 180,E1 -20743.218,E2 -20743.218} C_VEL
LIN {X 0,Y 225.376,Z 184.81,A -85,B 0,C 180,E1 -20745.122,E2 -20745.122} C_VEL
LIN {X 0,Y 233.468,Z 197.994,A -85,B 0,C 180,E1 -20747.439,E2 -20747.439} C_VEL
LIN {X 0,Y 237.72,Z 206.067,A -85,B 0,C 180,E1 -20748.607,E2 -20748.607} C_VEL
LIN {X 0,Y 242.134,Z 215.977,A -85,B 0,C 180,E1 -20749.814,E2 -20749.814} C_VEL
LIN {X 0,Y 239.74,Z 268.981,A -85,B 0,C 180,E1 -20751.369,E2 -20751.369} C_VEL
LIN {X 0,Y 238.493,Z 281.974,A -85,B 0,C 180,E1 -20752.036,E2 -20752.036} C_VEL
LIN {X 0,Y 236.594,Z 294.87,A -85,B 0,C 180,E1 -20753.02,E2 -20753.02} C_VEL
LIN {X 0,Y 234.603,Z 305.714,A -85,B 0,C 180,E1 -20754.166,E2 -20754.166} C_VEL
LIN {X 0,Y 232.067,Z 316.687,A -85,B 0,C 180,E1 -20755.663,E2 -20755.663} C_VEL
LIN {X 0,Y 229.063,Z 327.398,A -85,B 0,C 180,E1 -20757.524,E2 -20757.524} C_VEL
LIN {X 0,Y 226.011,Z 337.021,A -85,B 0,C 180,E1 -20759.647,E2 -20759.647} C_VEL
LIN {X 0,Y 223.385,Z 344.879,A -85,B 0,C 180,E1 -20761.84,E2 -20761.84} C_VEL
LIN {X 0,Y 220.585,Z 352.519,A -85,B 0,C 180,E1 -20764.523,E2 -20764.523} C_VEL
LIN {X 0,Y 218.063,Z 358.636,A -85,B 0,C 180,E1 -20767.246,E2 -20767.246} C_VEL
LIN {X 0,Y 216.003,Z 363.47,A -85,B 0,C 180,E1 -20770.022,E2 -20770.022} C_VEL
LIN {X 0,Y 214.355,Z 367.173,A -85,B 0,C 180,E1 -20772.836,E2 -20772.836} C_VEL
LIN {X 0,Y 213.496,Z 369.075,A -85,B 0,C 180,E1 -20774.73,E2 -20774.73} C_VEL
LIN {X 0,Y 212.791,Z 370.549,A -85,B 0,C 180,E1 -20776.631,E2 -20776.631} C_VEL
LIN {X 0,Y 211.99,Z 372.205,A -85,B 0,C 180,E1 -20780.457,E2 -20780.457} C_VEL
LIN {X 0,Y 211.847,Z 372.455,A -85,B 0,C 180,E1 -20782.373,E2 -20782.373} C_VEL
LIN {X 0,Y 211.766,Z 372.223,A -85,B 0,C 180,E1 -20784.646,E2 -20784.646} C_VEL
LIN {X 0,Y 211.768,Z 370.81,A -85,B 0,C 180,E1 -20788.096,E2 -20788.096} C_VEL
LIN {X 0,Y 211.872,Z 369.485,A -85,B 0,C 180,E1 -20789.998,E2 -20789.998} C_VEL
LIN {X 0,Y 212.369,Z 366.682,A -85,B 0,C 180,E1 -20792.844,E2 -20792.844} C_VEL
LIN {X 0,Y 213.148,Z 362.873,A -85,B 0,C 180,E1 -20795.675,E2 -20795.675} C_VEL
LIN {X 0,Y 214.37,Z 357.943,A -85,B 0,C 180,E1 -20798.482,E2 -20798.482} C_VEL
LIN {X 0,Y 215.829,Z 351.762,A -85,B 0,C 180,E1 -20801.265,E2 -20801.265} C_VEL
LIN {X 0,Y 217.945,Z 344.009,A -85,B 0,C 180,E1 -20803.994,E2 -20803.994} C_VEL
LIN {X 0,Y 220.002,Z 335.459,A -85,B 0,C 180,E1 -20806.406,E2 -20806.406} C_VEL
LIN {X 0,Y 222.259,Z 325.422,A -85,B 0,C 180,E1 -20808.671,E2 -20808.671} C_VEL
LIN {X 0,Y 224.469,Z 314.393,A -85,B 0,C 180,E1 -20810.622,E2 -20810.622} C_VEL
LIN {X 0,Y 226.633,Z 301.836,A -85,B 0,C 180,E1 -20812.324,E2 -20812.324} C_VEL
LIN {X 0,Y 228.086,Z 290.567,A -85,B 0,C 180,E1 -20813.491,E2 -20813.491} C_VEL
LIN {X 0,Y 229.346,Z 277.757,A -85,B 0,C 180,E1 -20814.435,E2 -20814.435} C_VEL
LIN {X 0,Y 230.2,Z 264.15,A -85,B 0,C 180,E1 -20815.06,E2 -20815.06} C_VEL
LIN {X 0,Y 232.422,Z 204.999,A -85,B 0,C 180,E1 -20816.822,E2 -20816.822} C_VEL
LIN {X 0,Y 227.682,Z 193.415,A -85,B 0,C 180,E1 -20817.926,E2 -20817.926} C_VEL
LIN {X 0,Y 220.679,Z 179.801,A -85,B 0,C 180,E1 -20819.538,E2 -20819.538} C_VEL
LIN {X 0,Y 215.375,Z 170.481,A -85,B 0,C 180,E1 -20820.809,E2 -20820.809} C_VEL
LIN {X 0,Y 214.008,Z 167.927,A -85,B 0,C 180,E1 -20821.157,E2 -20821.157} C_VEL
LIN {X 0,Y 213.795,Z 166.852,A -85,B 0,C 180,E1 -20821.274,E2 -20821.274} C_VEL
LIN {X 0,Y 213.781,Z 166.852,A -85,B 0,C 180,E1 -20824.727,E2 -20824.727} C_VEL
LIN {X 0,Y 213.731,Z 166.858,A -85,B 0,C 180,E1 -20828.662,E2 -20828.662} C_VEL
LIN {X 0,Y 213.701,Z 166.864,A -85,B 0,C 180,E1 -20833.677,E2 -20833.677} C_VEL
LIN {X 0,Y 213.701,Z 166.862,A -85,B 0,C 180,E1 -20836.342,E2 -20836.342} C_VEL
LIN {X 0,Y 213.712,Z 166.863,A -85,B 0,C 180,E1 -20839.141,E2 -20839.141} C_VEL
LIN {X 0,Y 213.738,Z 166.86,A -85,B 0,C 180,E1 -20843.71,E2 -20843.71} C_VEL
LIN {X 0,Y 213.774,Z 166.855,A -85,B 0,C 180,E1 -20848.73,E2 -20848.73} C_VEL
LIN {X 0,Y 213.819,Z 166.842,A -85,B 0,C 180,E1 -20852.602,E2 -20852.602} C_VEL
LIN {X 0,Y 213.811,Z 166.85,A -85,B 0,C 180,E1 -20856.973,E2 -20856.973} C_VEL
LIN {X 0,Y 213.883,Z 166.841,A -85,B 0,C 180,E1 -20862.798,E2 -20862.798} C_VEL
LIN {X 0,Y 213.924,Z 166.835,A -85,B 0,C 180,E1 -20866.704,E2 -20866.704} C_VEL
LIN {X 0,Y 214.124,Z 166.801,A -85,B 0,C 180,E1 -20870.554,E2 -20870.554} C_VEL
LIN {X 0,Y 214.061,Z 166.779,A -85,B 0,C 180,E1 -20874.347,E2 -20874.347} C_VEL
LIN {X 0,Y 214.393,Z 166.773,A -85,B 0,C 180,E1 -20878.121,E2 -20878.121} C_VEL
LIN {X 0,Y 214.501,Z 166.765,A -85,B 0,C 180,E1 -20880,E2 -20880} C_VEL
LIN {X 0,Y 214.394,Z 166.776,A -85,B 0,C 180,E1 -20881.878,E2 -20881.878} C_VEL
LIN {X 0,Y 214.167,Z 166.804,A -85,B 0,C 180,E1 -20887.542,E2 -20887.542} C_VEL
LIN {X 0,Y 213.983,Z 166.827,A -85,B 0,C 180,E1 -20891.365,E2 -20891.365} C_VEL
LIN {X 0,Y 213.89,Z 166.842,A -85,B 0,C 180,E1 -20895.24,E2 -20895.24} C_VEL
LIN {X 0,Y 213.803,Z 166.855,A -85,B 0,C 180,E1 -20899.191,E2 -20899.191} C_VEL
LIN {X 0,Y 213.802,Z 166.856,A -85,B 0,C 180,E1 -20903.232,E2 -20903.232} C_VEL
LIN {X 0,Y 213.822,Z 166.853,A -85,B 0,C 180,E1 -20907.451,E2 -20907.451} C_VEL
LIN {X 0,Y 213.76,Z 166.861,A -85,B 0,C 180,E1 -20911.739,E2 -20911.739} C_VEL
LIN {X 0,Y 213.737,Z 166.865,A -85,B 0,C 180,E1 -20916.29,E2 -20916.29} C_VEL
LIN {X 0,Y 213.706,Z 166.865,A -85,B 0,C 180,E1 -20921.127,E2 -20921.127} C_VEL
LIN {X 0,Y 213.665,Z 166.865,A -85,B 0,C 180,E1 -20925.817,E2 -20925.817} C_VEL
LIN {X 0,Y 213.111,Z 167.263,A -85,B 0,C 180,E1 -20926.871,E2 -20926.871} C_VEL
LIN {X 0,Y 211.252,Z 168.718,A -85,B 0,C 180,E1 -20928.184,E2 -20928.184} C_VEL
LIN {X 0,Y 208.54,Z 172.14,A -85,B 0,C 180,E1 -20930.087,E2 -20930.087} C_VEL
LIN {X 0,Y 208.353,Z 174.123,A -85,B 0,C 180,E1 -20931.061,E2 -20931.061} C_VEL
LIN {X 0,Y 209.304,Z 177.745,A -85,B 0,C 180,E1 -20932.758,E2 -20932.758} C_VEL
LIN {X 0,Y 216.722,Z 193.997,A -85,B 0,C 180,E1 -20934.732,E2 -20934.732} C_VEL
LIN {X 0,Y 221.755,Z 206.987,A -85,B 0,C 180,E1 -20936.047,E2 -20936.047} C_VEL
LIN {X 0,Y 224.725,Z 233.004,A -85,B 0,C 180,E1 -20937.453,E2 -20937.453} C_VEL
LIN {X 0,Y 225.025,Z 237.802,A -85,B 0,C 180,E1 -20937.67,E2 -20937.67} C_VEL
LIN {X 0,Y 223.008,Z 287.708,A -85,B 0,C 180,E1 -20939.24,E2 -20939.24} C_VEL
LIN {X 0,Y 221.803,Z 301.062,A -85,B 0,C 180,E1 -20940,E2 -20940} C_VEL
LIN {X 0,Y 220.142,Z 313.051,A -85,B 0,C 180,E1 -20940.999,E2 -20940.999} C_VEL
LIN {X 0,Y 218.016,Z 325.172,A -85,B 0,C 180,E1 -20942.396,E2 -20942.396} C_VEL
LIN {X 0,Y 215.639,Z 336.729,A -85,B 0,C 180,E1 -20944.159,E2 -20944.159} C_VEL
LIN {X 0,Y 213.181,Z 347.138,A -85,B 0,C 180,E1 -20946.183,E2 -20946.183} C_VEL
LIN {X 0,Y 210.912,Z 356.491,A -85,B 0,C 180,E1 -20948.5,E2 -20948.5} C_VEL
LIN {X 0,Y 208.829,Z 365.578,A -85,B 0,C 180,E1 -20951.356,E2 -20951.356} C_VEL
LIN {X 0,Y 206.999,Z 372.88,A -85,B 0,C 180,E1 -20954.242,E2 -20954.242} C_VEL
LIN {X 0,Y 205.644,Z 378.716,A -85,B 0,C 180,E1 -20957.167,E2 -20957.167} C_VEL
LIN {X 0,Y 204.879,Z 383.315,A -85,B 0,C 180,E1 -20960.126,E2 -20960.126} C_VEL
LIN {X 0,Y 204.619,Z 385.738,A -85,B 0,C 180,E1 -20962.105,E2 -20962.105} C_VEL
LIN {X 0,Y 204.466,Z 388.808,A -85,B 0,C 180,E1 -20965.418,E2 -20965.418} C_VEL
LIN {X 0,Y 204.554,Z 390.397,A -85,B 0,C 180,E1 -20968.033,E2 -20968.033} C_VEL
LIN {X 0,Y 204.67,Z 391.091,A -85,B 0,C 180,E1 -20970.002,E2 -20970.002} C_VEL
LIN {X 0,Y 204.528,Z 391.378,A -85,B 0,C 180,E1 -20971.971,E2 -20971.971} C_VEL
LIN {X 0,Y 204.412,Z 391.188,A -85,B 0,C 180,E1 -20974.389,E2 -20974.389} C_VEL
LIN {X 0,Y 204.567,Z 389.821,A -85,B 0,C 180,E1 -20977.9,E2 -20977.9} C_VEL
LIN {X 0,Y 204.945,Z 388.498,A -85,B 0,C 180,E1 -20979.874,E2 -20979.874} C_VEL
LIN {X 0,Y 205.807,Z 385.719,A -85,B 0,C 180,E1 -20982.826,E2 -20982.826} C_VEL
LIN {X 0,Y 207.238,Z 381.935,A -85,B 0,C 180,E1 -20985.743,E2 -20985.743} C_VEL
LIN {X 0,Y 209.232,Z 377.047,A -85,B 0,C 180,E1 -20988.61,E2 -20988.61} C_VEL
LIN {X 0,Y 211.647,Z 370.906,A -85,B 0,C 180,E1 -20991.426,E2 -20991.426} C_VEL
LIN {X 0,Y 214.477,Z 363.295,A -85,B 0,C 180,E1 -20994.181,E2 -20994.181} C_VEL
LIN {X 0,Y 217.408,Z 355.534,A -85,B 0,C 180,E1 -20996.392,E2 -20996.392} C_VEL
LIN {X 0,Y 221.013,Z 345.007,A -85,B 0,C 180,E1 -20998.75,E2 -20998.75} C_VEL
LIN {X 0,Y 224.3,Z 334.311,A -85,B 0,C 180,E1 -21000.609,E2 -21000.609} C_VEL
LIN {X 0,Y 227.067,Z 323.964,A -85,B 0,C 180,E1 -21002.01,E2 -21002.01} C_VEL
LIN {X 0,Y 229.77,Z 311.572,A -85,B 0,C 180,E1 -21003.276,E2 -21003.276} C_VEL
LIN {X 0,Y 231.922,Z 298.532,A -85,B 0,C 180,E1 -21004.231,E2 -21004.231} C_VEL
LIN {X 0,Y 233.243,Z 285.74,A -85,B 0,C 180,E1 -21004.86,E2 -21004.86} C_VEL
LIN {X 0,Y 235.393,Z 240.913,A -85,B 0,C 180,E1 -21006.191,E2 -21006.191} C_VEL
LIN {X 0,Y 232.846,Z 222.51,A -85,B 0,C 180,E1 -21007.401,E2 -21007.401} C_VEL
LIN {X 0,Y 226.349,Z 207.585,A -85,B 0,C 180,E1 -21009.378,E2 -21009.378} C_VEL
LIN {X 0,Y 220.317,Z 195.507,A -85,B 0,C 180,E1 -21011.301,E2 -21011.301} C_VEL
LIN {X 0,Y 215.023,Z 186.136,A -85,B 0,C 180,E1 -21013.077,E2 -21013.077} C_VEL
LIN {X 0,Y 211.961,Z 181.045,A -85,B 0,C 180,E1 -21014.156,E2 -21014.156} C_VEL
LIN {X 0,Y 209.152,Z 176.184,A -85,B 0,C 180,E1 -21015.275,E2 -21015.275} C_VEL
LIN {X 0,Y 207.525,Z 170.584,A -85,B 0,C 180,E1 -21018.731,E2 -21018.731} C_VEL
LIN {X 0,Y 206.662,Z 167.742,A -85,B 0,C 180,E1 -21020.691,E2 -21020.691} C_VEL
LIN {X 0,Y 206.703,Z 167.737,A -85,B 0,C 180,E1 -21024.689,E2 -21024.689} C_VEL
LIN {X 0,Y 206.699,Z 167.736,A -85,B 0,C 180,E1 -21029.335,E2 -21029.335} C_VEL
LIN {X 0,Y 206.707,Z 167.734,A -85,B 0,C 180,E1 -21033.769,E2 -21033.769} C_VEL
LIN {X 0,Y 206.72,Z 167.735,A -85,B 0,C 180,E1 -21038.039,E2 -21038.039} C_VEL
LIN {X 0,Y 206.806,Z 167.719,A -85,B 0,C 180,E1 -21042.191,E2 -21042.191} C_VEL
LIN {X 0,Y 206.852,Z 167.702,A -85,B 0,C 180,E1 -21046.242,E2 -21046.242} C_VEL
LIN {X 0,Y 207.075,Z 167.679,A -85,B 0,C 180,E1 -21050.23,E2 -21050.23} C_VEL
LIN {X 0,Y 207.032,Z 167.697,A -85,B 0,C 180,E1 -21054.155,E2 -21054.155} C_VEL
LIN {X 0,Y 207.32,Z 167.645,A -85,B 0,C 180,E1 -21058.058,E2 -21058.058} C_VEL
LIN {X 0,Y 207.479,Z 167.642,A -85,B 0,C 180,E1 -21060,E2 -21060} C_VEL
LIN {X 0,Y 207.343,Z 167.644,A -85,B 0,C 180,E1 -21061.943,E2 -21061.943} C_VEL
LIN {X 0,Y 207.128,Z 167.67,A -85,B 0,C 180,E1 -21067.801,E2 -21067.801} C_VEL
LIN {X 0,Y 206.916,Z 167.711,A -85,B 0,C 180,E1 -21071.759,E2 -21071.759} C_VEL
LIN {X 0,Y 206.818,Z 167.715,A -85,B 0,C 180,E1 -21075.775,E2 -21075.775} C_VEL
LIN {X 0,Y 206.72,Z 167.721,A -85,B 0,C 180,E1 -21079.876,E2 -21079.876} C_VEL
LIN {X 0,Y 206.738,Z 167.72,A -85,B 0,C 180,E1 -21084.076,E2 -21084.076} C_VEL
LIN {X 0,Y 206.693,Z 167.729,A -85,B 0,C 180,E1 -21088.427,E2 -21088.427} C_VEL
LIN {X 0,Y 206.699,Z 167.729,A -85,B 0,C 180,E1 -21092.958,E2 -21092.958} C_VEL
LIN {X 0,Y 206.68,Z 167.738,A -85,B 0,C 180,E1 -21097.74,E2 -21097.74} C_VEL
LIN {X 0,Y 206.649,Z 167.728,A -85,B 0,C 180,E1 -21099.255,E2 -21099.255} C_VEL
LIN {X 0,Y 207.536,Z 170.398,A -85,B 0,C 180,E1 -21099.696,E2 -21099.696} C_VEL
LIN {X 0,Y 209.61,Z 172.649,A -85,B 0,C 180,E1 -21100.433,E2 -21100.433} C_VEL
LIN {X 0,Y 212.398,Z 176.741,A -85,B 0,C 180,E1 -21101.436,E2 -21101.436} C_VEL
LIN {X 0,Y 219.053,Z 186.383,A -85,B 0,C 180,E1 -21103.656,E2 -21103.656} C_VEL
LIN {X 0,Y 227.343,Z 199.656,A -85,B 0,C 180,E1 -21106.191,E2 -21106.191} C_VEL
LIN {X 0,Y 232.787,Z 209.788,A -85,B 0,C 180,E1 -21107.763,E2 -21107.763} C_VEL
LIN {X 0,Y 236.475,Z 218.208,A -85,B 0,C 180,E1 -21108.828,E2 -21108.828} C_VEL
LIN {X 0,Y 234.053,Z 269.227,A -85,B 0,C 180,E1 -21110.35,E2 -21110.35} C_VEL
LIN {X 0,Y 232.688,Z 282.653,A -85,B 0,C 180,E1 -21111.051,E2 -21111.051} C_VEL
LIN {X 0,Y 230.739,Z 295.46,A -85,B 0,C 180,E1 -21112.055,E2 -21112.055} C_VEL
LIN {X 0,Y 228.619,Z 306.43,A -85,B 0,C 180,E1 -21113.244,E2 -21113.244} C_VEL
LIN {X 0,Y 225.843,Z 317.81,A -85,B 0,C 180,E1 -21114.85,E2 -21114.85} C_VEL
LIN {X 0,Y 222.715,Z 328.383,A -85,B 0,C 180,E1 -21116.749,E2 -21116.749} C_VEL
LIN {X 0,Y 219.86,Z 337.003,A -85,B 0,C 180,E1 -21118.704,E2 -21118.704} C_VEL
LIN {X 0,Y 217.094,Z 344.922,A -85,B 0,C 180,E1 -21120.947,E2 -21120.947} C_VEL
LIN {X 0,Y 214.149,Z 352.63,A -85,B 0,C 180,E1 -21123.7,E2 -21123.7} C_VEL
LIN {X 0,Y 211.467,Z 358.788,A -85,B 0,C 180,E1 -21126.494,E2 -21126.494} C_VEL
LIN {X 0,Y 209.276,Z 363.659,A -85,B 0,C 180,E1 -21129.351,E2 -21129.351} C_VEL
LIN {X 0,Y 207.522,Z 367.396,A -85,B 0,C 180,E1 -21132.252,E2 -21132.252} C_VEL
LIN {X 0,Y 206.598,Z 369.315,A -85,B 0,C 180,E1 -21134.207,E2 -21134.207} C_VEL
LIN {X 0,Y 205.828,Z 370.815,A -85,B 0,C 180,E1 -21136.17,E2 -21136.17} C_VEL
LIN {X 0,Y 204.935,Z 372.508,A -85,B 0,C 180,E1 -21140.125,E2 -21140.125} C_VEL
LIN {X 0,Y 204.762,Z 372.773,A -85,B 0,C 180,E1 -21142.107,E2 -21142.107} C_VEL
LIN {X 0,Y 204.68,Z 372.504,A -85,B 0,C 180,E1 -21144.726,E2 -21144.726} C_VEL
LIN {X 0,Y 204.677,Z 371.188,A -85,B 0,C 180,E1 -21148.03,E2 -21148.03} C_VEL
LIN {X 0,Y 204.8,Z 369.877,A -85,B 0,C 180,E1 -21149.998,E2 -21149.998} C_VEL
LIN {X 0,Y 205.297,Z 367.106,A -85,B 0,C 180,E1 -21152.942,E2 -21152.942} C_VEL
LIN {X 0,Y 206.106,Z 363.331,A -85,B 0,C 180,E1 -21155.87,E2 -21155.87} C_VEL
LIN {X 0,Y 207.367,Z 358.439,A -85,B 0,C 180,E1 -21158.771,E2 -21158.771} C_VEL
LIN {X 0,Y 208.908,Z 352.296,A -85,B 0,C 180,E1 -21161.643,E2 -21161.643} C_VEL
LIN {X 0,Y 211.102,Z 344.614,A -85,B 0,C 180,E1 -21164.457,E2 -21164.457} C_VEL
LIN {X 0,Y 213.505,Z 335.008,A -85,B 0,C 180,E1 -21167.231,E2 -21167.231} C_VEL
LIN {X 0,Y 215.831,Z 325.084,A -85,B 0,C 180,E1 -21169.495,E2 -21169.495} C_VEL
LIN {X 0,Y 218.148,Z 313.843,A -85,B 0,C 180,E1 -21171.496,E2 -21171.496} C_VEL
LIN {X 0,Y 220.127,Z 302.83,A -85,B 0,C 180,E1 -21173.021,E2 -21173.021} C_VEL
LIN {X 0,Y 221.783,Z 290.621,A -85,B 0,C 180,E1 -21174.325,E2 -21174.325} C_VEL
LIN {X 0,Y 223.118,Z 277.652,A -85,B 0,C 180,E1 -21175.288,E2 -21175.288} C_VEL
LIN {X 0,Y 223.998,Z 263.776,A -85,B 0,C 180,E1 -21175.929,E2 -21175.929} C_VEL
LIN {X 0,Y 226.315,Z 207.15,A -85,B 0,C 180,E1 -21177.636,E2 -21177.636} C_VEL
LIN {X 0,Y 222.409,Z 197.385,A -85,B 0,C 180,E1 -21178.598,E2 -21178.598} C_VEL
LIN {X 0,Y 215.763,Z 184.208,A -85,B 0,C 180,E1 -21180.203,E2 -21180.203} C_VEL
LIN {X 0,Y 208.555,Z 171.685,A -85,B 0,C 180,E1 -21182.025,E2 -21182.025} C_VEL
LIN {X 0,Y 207.069,Z 169.232,A -85,B 0,C 180,E1 -21182.416,E2 -21182.416} C_VEL
LIN {X 0,Y 206.709,Z 167.733,A -85,B 0,C 180,E1 -21182.58,E2 -21182.58} C_VEL
LIN {X 0,Y 206.719,Z 167.732,A -85,B 0,C 180,E1 -21185.318,E2 -21185.318} C_VEL
LIN {X 0,Y 206.659,Z 167.741,A -85,B 0,C 180,E1 -21190.249,E2 -21190.249} C_VEL
LIN {X 0,Y 206.628,Z 167.748,A -85,B 0,C 180,E1 -21195.58,E2 -21195.58} C_VEL
LIN {X 0,Y 206.655,Z 167.745,A -85,B 0,C 180,E1 -21199.747,E2 -21199.747} C_VEL
LIN {X 0,Y 206.693,Z 167.739,A -85,B 0,C 180,E1 -21204.687,E2 -21204.687} C_VEL
LIN {X 0,Y 206.7,Z 167.738,A -85,B 0,C 180,E1 -21209.335,E2 -21209.335} C_VEL
LIN {X 0,Y 206.723,Z 167.731,A -85,B 0,C 180,E1 -21213.77,E2 -21213.77} C_VEL
LIN {X 0,Y 206.723,Z 167.725,A -85,B 0,C 180,E1 -21218.039,E2 -21218.039} C_VEL
LIN {X 0,Y 206.816,Z 167.721,A -85,B 0,C 180,E1 -21222.191,E2 -21222.191} C_VEL
LIN {X 0,Y 206.865,Z 167.714,A -85,B 0,C 180,E1 -21226.242,E2 -21226.242} C_VEL
LIN {X 0,Y 207.069,Z 167.683,A -85,B 0,C 180,E1 -21230.229,E2 -21230.229} C_VEL
LIN {X 0,Y 207.025,Z 167.653,A -85,B 0,C 180,E1 -21234.154,E2 -21234.154} C_VEL
LIN {X 0,Y 207.333,Z 167.652,A -85,B 0,C 180,E1 -21238.057,E2 -21238.057} C_VEL
LIN {X 0,Y 207.469,Z 167.641,A -85,B 0,C 180,E1 -21240,E2 -21240} C_VEL
LIN {X 0,Y 207.334,Z 167.655,A -85,B 0,C 180,E1 -21241.942,E2 -21241.942} C_VEL
LIN {X 0,Y 207.112,Z 167.683,A -85,B 0,C 180,E1 -21247.801,E2 -21247.801} C_VEL
LIN {X 0,Y 206.905,Z 167.708,A -85,B 0,C 180,E1 -21251.759,E2 -21251.759} C_VEL
LIN {X 0,Y 206.818,Z 167.722,A -85,B 0,C 180,E1 -21255.774,E2 -21255.774} C_VEL
LIN {X 0,Y 206.738,Z 167.734,A -85,B 0,C 180,E1 -21259.873,E2 -21259.873} C_VEL
LIN {X 0,Y 206.738,Z 167.736,A -85,B 0,C 180,E1 -21264.075,E2 -21264.075} C_VEL
LIN {X 0,Y 206.729,Z 167.735,A -85,B 0,C 180,E1 -21268.421,E2 -21268.421} C_VEL
LIN {X 0,Y 206.692,Z 167.742,A -85,B 0,C 180,E1 -21272.959,E2 -21272.959} C_VEL
LIN {X 0,Y 206.673,Z 167.744,A -85,B 0,C 180,E1 -21277.741,E2 -21277.741} C_VEL
LIN {X 0,Y 206.636,Z 167.747,A -85,B 0,C 180,E1 -21281.564,E2 -21281.564} C_VEL
LIN {X 0,Y 206.621,Z 167.745,A -85,B 0,C 180,E1 -21285.807,E2 -21285.807} C_VEL
LIN {X 0,Y 206.686,Z 167.815,A -85,B 0,C 180,E1 -21287.876,E2 -21287.876} C_VEL
LIN {X 0,Y 208.353,Z 174.123,A -85,B 0,C 180,E1 -21291.061,E2 -21291.061} C_VEL
LIN {X 0,Y 208.834,Z 176.523,A -85,B 0,C 180,E1 -21291.874,E2 -21291.874} C_VEL
LIN {X 0,Y 209.41,Z 180.509,A -85,B 0,C 180,E1 -21292.62,E2 -21292.62} C_VEL
LIN {X 0,Y 210.159,Z 186.966,A -85,B 0,C 180,E1 -21293.293,E2 -21293.293} C_VEL
LIN {X 0,Y 211.3,Z 195.043,A -85,B 0,C 180,E1 -21293.826,E2 -21293.826} C_VEL
LIN {X 0,Y 212.707,Z 200.852,A -85,B 0,C 180,E1 -21294.305,E2 -21294.305} C_VEL
LIN {X 0,Y 213.419,Z 202.66,A -85,B 0,C 180,E1 -21294.502,E2 -21294.502} C_VEL
LIN {X 0,Y 215.994,Z 209.89,A -85,B 0,C 180,E1 -21295.222,E2 -21295.222} C_VEL
LIN {X 0,Y 218.925,Z 237.511,A -85,B 0,C 180,E1 -21296.742,E2 -21296.742} C_VEL
LIN {X 0,Y 216.778,Z 287.417,A -85,B 0,C 180,E1 -21298.344,E2 -21298.344} C_VEL
LIN {X 0,Y 215.566,Z 300.536,A -85,B 0,C 180,E1 -21299.106,E2 -21299.106} C_VEL
LIN {X 0,Y 213.753,Z 313.139,A -85,B 0,C 180,E1 -21300.181,E2 -21300.181} C_VEL
LIN {X 0,Y 211.704,Z 324.343,A -85,B 0,C 180,E1 -21301.499,E2 -21301.499} C_VEL
LIN {X 0,Y 209.227,Z 335.993,A -85,B 0,C 180,E1 -21303.305,E2 -21303.305} C_VEL
LIN {X 0,Y 206.679,Z 346.475,A -85,B 0,C 180,E1 -21305.385,E2 -21305.385} C_VEL
LIN {X 0,Y 204.286,Z 355.908,A -85,B 0,C 180,E1 -21307.766,E2 -21307.766} C_VEL
LIN {X 0,Y 202.4,Z 363.665,A -85,B 0,C 180,E1 -21310.214,E2 -21310.214} C_VEL
LIN {X 0,Y 200.434,Z 371.25,A -85,B 0,C 180,E1 -21313.187,E2 -21313.187} C_VEL
LIN {X 0,Y 198.665,Z 378.253,A -85,B 0,C 180,E1 -21316.708,E2 -21316.708} C_VEL
LIN {X 0,Y 197.86,Z 382.886,A -85,B 0,C 180,E1 -21319.772,E2 -21319.772} C_VEL
LIN {X 0,Y 197.562,Z 385.329,A -85,B 0,C 180,E1 -21321.821,E2 -21321.821} C_VEL
LIN {X 0,Y 197.371,Z 388.662,A -85,B 0,C 180,E1 -21325.581,E2 -21325.581} C_VEL
LIN {X 0,Y 197.469,Z 390.042,A -85,B 0,C 180,E1 -21327.962,E2 -21327.962} C_VEL
LIN {X 0,Y 197.581,Z 390.748,A -85,B 0,C 180,E1 -21330.002,E2 -21330.002} C_VEL
LIN {X 0,Y 197.44,Z 391.048,A -85,B 0,C 180,E1 -21332.042,E2 -21332.042} C_VEL
LIN {X 0,Y 197.338,Z 390.935,A -85,B 0,C 180,E1 -21334.293,E2 -21334.293} C_VEL
LIN {X 0,Y 197.507,Z 389.54,A -85,B 0,C 180,E1 -21338.185,E2 -21338.185} C_VEL
LIN {X 0,Y 197.926,Z 388.23,A -85,B 0,C 180,E1 -21340.228,E2 -21340.228} C_VEL
LIN {X 0,Y 198.849,Z 385.477,A -85,B 0,C 180,E1 -21343.283,E2 -21343.283} C_VEL
LIN {X 0,Y 200.383,Z 381.722,A -85,B 0,C 180,E1 -21346.297,E2 -21346.297} C_VEL
LIN {X 0,Y 202.486,Z 376.864,A -85,B 0,C 180,E1 -21349.254,E2 -21349.254} C_VEL
LIN {X 0,Y 205.201,Z 370.252,A -85,B 0,C 180,E1 -21352.372,E2 -21352.372} C_VEL
LIN {X 0,Y 208.002,Z 363.184,A -85,B 0,C 180,E1 -21354.985,E2 -21354.985} C_VEL
LIN {X 0,Y 211.083,Z 355.472,A -85,B 0,C 180,E1 -21357.247,E2 -21357.247} C_VEL
LIN {X 0,Y 214.459,Z 346.089,A -85,B 0,C 180,E1 -21359.445,E2 -21359.445} C_VEL
LIN {X 0,Y 217.845,Z 335.686,A -85,B 0,C 180,E1 -21361.348,E2 -21361.348} C_VEL
LIN {X 0,Y 221.079,Z 324.143,A -85,B 0,C 180,E1 -21362.985,E2 -21362.985} C_VEL
LIN {X 0,Y 223.891,Z 311.965,A -85,B 0,C 180,E1 -21364.269,E2 -21364.269} C_VEL
LIN {X 0,Y 226.095,Z 299.177,A -85,B 0,C 180,E1 -21365.241,E2 -21365.241} C_VEL
LIN {X 0,Y 227.596,Z 285.783,A -85,B 0,C 180,E1 -21365.925,E2 -21365.925} C_VEL
LIN {X 0,Y 229.822,Z 242.233,A -85,B 0,C 180,E1 -21367.238,E2 -21367.238} C_VEL
LIN {X 0,Y 227.668,Z 225.611,A -85,B 0,C 180,E1 -21368.352,E2 -21368.352} C_VEL
LIN {X 0,Y 221.541,Z 211.35,A -85,B 0,C 180,E1 -21370.32,E2 -21370.32} C_VEL
LIN {X 0,Y 215.967,Z 199.993,A -85,B 0,C 180,E1 -21372.193,E2 -21372.193} C_VEL
LIN {X 0,Y 210.8,Z 190.712,A -85,B 0,C 180,E1 -21374.019,E2 -21374.019} C_VEL
LIN {X 0,Y 207.96,Z 185.933,A -85,B 0,C 180,E1 -21375.072,E2 -21375.072} C_VEL
LIN {X 0,Y 204.673,Z 180.65,A -85,B 0,C 180,E1 -21376.344,E2 -21376.344} C_VEL
LIN {X 0,Y 201.947,Z 176.186,A -85,B 0,C 180,E1 -21377.46,E2 -21377.46} C_VEL
LIN {X 0,Y 201.765,Z 175.769,A -85,B 0,C 180,E1 -21377.573,E2 -21377.573} C_VEL
LIN {X 0,Y 199.631,Z 168.618,A -85,B 0,C 180,E1 -21382.527,E2 -21382.527} C_VEL
LIN {X 0,Y 199.689,Z 168.613,A -85,B 0,C 180,E1 -21388.135,E2 -21388.135} C_VEL
LIN {X 0,Y 199.646,Z 168.617,A -85,B 0,C 180,E1 -21392.766,E2 -21392.766} C_VEL
LIN {X 0,Y 199.681,Z 168.61,A -85,B 0,C 180,E1 -21397.222,E2 -21397.222} C_VEL
LIN {X 0,Y 199.749,Z 168.593,A -85,B 0,C 180,E1 -21401.803,E2 -21401.803} C_VEL
LIN {X 0,Y 199.77,Z 168.583,A -85,B 0,C 180,E1 -21405.744,E2 -21405.744} C_VEL
LIN {X 0,Y 200.027,Z 168.56,A -85,B 0,C 180,E1 -21409.882,E2 -21409.882} C_VEL
LIN {X 0,Y 199.996,Z 168.572,A -85,B 0,C 180,E1 -21413.949,E2 -21413.949} C_VEL
LIN {X 0,Y 200.265,Z 168.523,A -85,B 0,C 180,E1 -21417.989,E2 -21417.989} C_VEL
LIN {X 0,Y 200.446,Z 168.518,A -85,B 0,C 180,E1 -21420,E2 -21420} C_VEL
LIN {X 0,Y 199.985,Z 168.56,A -85,B 0,C 180,E1 -21424.031,E2 -21424.031} C_VEL
LIN {X 0,Y 200.076,Z 168.546,A -85,B 0,C 180,E1 -21428.077,E2 -21428.077} C_VEL
LIN {X 0,Y 199.865,Z 168.587,A -85,B 0,C 180,E1 -21432.18,E2 -21432.18} C_VEL
LIN {X 0,Y 199.759,Z 168.601,A -85,B 0,C 180,E1 -21436.348,E2 -21436.348} C_VEL
LIN {X 0,Y 199.653,Z 168.605,A -85,B 0,C 180,E1 -21440.611,E2 -21440.611} C_VEL
LIN {X 0,Y 199.653,Z 168.604,A -85,B 0,C 180,E1 -21444.987,E2 -21444.987} C_VEL
LIN {X 0,Y 199.613,Z 168.612,A -85,B 0,C 180,E1 -21449.533,E2 -21449.533} C_VEL
LIN {X 0,Y 199.67,Z 168.605,A -85,B 0,C 180,E1 -21452.352,E2 -21452.352} C_VEL
LIN {X 0,Y 199.605,Z 168.625,A -85,B 0,C 180,E1 -21457.004,E2 -21457.004} C_VEL
LIN {X 0,Y 200.474,Z 171.183,A -85,B 0,C 180,E1 -21457.447,E2 -21457.447} C_VEL
LIN {X 0,Y 202.44,Z 173.433,A -85,B 0,C 180,E1 -21458.231,E2 -21458.231} C_VEL
LIN {X 0,Y 203.165,Z 174.218,A -85,B 0,C 180,E1 -21458.512,E2 -21458.512} C_VEL
LIN {X 0,Y 205.311,Z 177.544,A -85,B 0,C 180,E1 -21459.372,E2 -21459.372} C_VEL
LIN {X 0,Y 206.766,Z 179.253,A -85,B 0,C 180,E1 -21459.909,E2 -21459.909} C_VEL
LIN {X 0,Y 214.951,Z 191.212,A -85,B 0,C 180,E1 -21462.814,E2 -21462.814} C_VEL
LIN {X 0,Y 223.12,Z 204.572,A -85,B 0,C 180,E1 -21465.436,E2 -21465.436} C_VEL
LIN {X 0,Y 228.044,Z 213.909,A -85,B 0,C 180,E1 -21466.929,E2 -21466.929} C_VEL
LIN {X 0,Y 230.951,Z 220.625,A -85,B 0,C 180,E1 -21467.813,E2 -21467.813} C_VEL
LIN {X 0,Y 228.346,Z 270.331,A -85,B 0,C 180,E1 -21469.312,E2 -21469.312} C_VEL
LIN {X 0,Y 226.855,Z 284.115,A -85,B 0,C 180,E1 -21470.067,E2 -21470.067} C_VEL
LIN {X 0,Y 224.955,Z 296.058,A -85,B 0,C 180,E1 -21471.041,E2 -21471.041} C_VEL
LIN {X 0,Y 222.442,Z 308.11,A -85,B 0,C 180,E1 -21472.397,E2 -21472.397} C_VEL
LIN {X 0,Y 219.288,Z 320.234,A -85,B 0,C 180,E1 -21474.203,E2 -21474.203} C_VEL
LIN {X 0,Y 216.086,Z 330.405,A -85,B 0,C 180,E1 -21476.152,E2 -21476.152} C_VEL
LIN {X 0,Y 213.157,Z 338.724,A -85,B 0,C 180,E1 -21478.159,E2 -21478.159} C_VEL
LIN {X 0,Y 209.691,Z 347.954,A -85,B 0,C 180,E1 -21481.011,E2 -21481.011} C_VEL
LIN {X 0,Y 206.724,Z 354.971,A -85,B 0,C 180,E1 -21483.769,E2 -21483.769} C_VEL
LIN {X 0,Y 204.1,Z 360.734,A -85,B 0,C 180,E1 -21486.671,E2 -21486.671} C_VEL
LIN {X 0,Y 201.441,Z 366.192,A -85,B 0,C 180,E1 -21490.391,E2 -21490.391} C_VEL
LIN {X 0,Y 199.724,Z 369.555,A -85,B 0,C 180,E1 -21493.648,E2 -21493.648} C_VEL
LIN {X 0,Y 198.88,Z 371.076,A -85,B 0,C 180,E1 -21495.677,E2 -21495.677} C_VEL
LIN {X 0,Y 198.316,Z 372.146,A -85,B 0,C 180,E1 -21497.722,E2 -21497.722} C_VEL
LIN {X 0,Y 197.689,Z 373.091,A -85,B 0,C 180,E1 -21501.823,E2 -21501.823} C_VEL
LIN {X 0,Y 197.604,Z 372.791,A -85,B 0,C 180,E1 -21504.785,E2 -21504.785} C_VEL
LIN {X 0,Y 197.588,Z 371.565,A -85,B 0,C 180,E1 -21507.96,E2 -21507.96} C_VEL
LIN {X 0,Y 197.728,Z 370.268,A -85,B 0,C 180,E1 -21509.998,E2 -21509.998} C_VEL
LIN {X 0,Y 198.227,Z 367.53,A -85,B 0,C 180,E1 -21513.047,E2 -21513.047} C_VEL
LIN {X 0,Y 199.068,Z 363.79,A -85,B 0,C 180,E1 -21516.078,E2 -21516.078} C_VEL
LIN {X 0,Y 200.372,Z 358.934,A -85,B 0,C 180,E1 -21519.079,E2 -21519.079} C_VEL
LIN {X 0,Y 201.998,Z 352.831,A -85,B 0,C 180,E1 -21522.047,E2 -21522.047} C_VEL
LIN {X 0,Y 204.273,Z 345.217,A -85,B 0,C 180,E1 -21524.951,E2 -21524.951} C_VEL
LIN {X 0,Y 206.398,Z 337.153,A -85,B 0,C 180,E1 -21527.414,E2 -21527.414} C_VEL
LIN {X 0,Y 208.947,Z 326.879,A -85,B 0,C 180,E1 -21529.909,E2 -21529.909} C_VEL
LIN {X 0,Y 211.343,Z 316.109,A -85,B 0,C 180,E1 -21531.967,E2 -21531.967} C_VEL
LIN {X 0,Y 213.665,Z 303.823,A -85,B 0,C 180,E1 -21533.76,E2 -21533.76} C_VEL
LIN {X 0,Y 215.388,Z 291.811,A -85,B 0,C 180,E1 -21535.097,E2 -21535.097} C_VEL
LIN {X 0,Y 216.75,Z 279.375,A -85,B 0,C 180,E1 -21536.086,E2 -21536.086} C_VEL
LIN {X 0,Y 217.699,Z 266.387,A -85,B 0,C 180,E1 -21536.738,E2 -21536.738} C_VEL
LIN {X 0,Y 220.098,Z 208.577,A -85,B 0,C 180,E1 -21538.548,E2 -21538.548} C_VEL
LIN {X 0,Y 216.484,Z 199.897,A -85,B 0,C 180,E1 -21539.471,E2 -21539.471} C_VEL
LIN {X 0,Y 209.569,Z 186.244,A -85,B 0,C 180,E1 -21541.237,E2 -21541.237} C_VEL
LIN {X 0,Y 203.167,Z 175.379,A -85,B 0,C 180,E1 -21542.938,E2 -21542.938} C_VEL
LIN {X 0,Y 201.369,Z 172.44,A -85,B 0,C 180,E1 -21543.438,E2 -21543.438} C_VEL
LIN {X 0,Y 199.911,Z 169.892,A -85,B 0,C 180,E1 -21543.859,E2 -21543.859} C_VEL
LIN {X 0,Y 199.638,Z 168.613,A -85,B 0,C 180,E1 -21544.019,E2 -21544.019} C_VEL
LIN {X 0,Y 199.636,Z 168.613,A -85,B 0,C 180,E1 -21546.757,E2 -21546.757} C_VEL
LIN {X 0,Y 199.635,Z 168.614,A -85,B 0,C 180,E1 -21549.319,E2 -21549.319} C_VEL
LIN {X 0,Y 199.575,Z 168.625,A -85,B 0,C 180,E1 -21554.769,E2 -21554.769} C_VEL
LIN {X 0,Y 199.574,Z 168.62,A -85,B 0,C 180,E1 -21558.003,E2 -21558.003} C_VEL
LIN {X 0,Y 199.605,Z 168.62,A -85,B 0,C 180,E1 -21560.766,E2 -21560.766} C_VEL
LIN {X 0,Y 199.606,Z 168.619,A -85,B 0,C 180,E1 -21565.712,E2 -21565.712} C_VEL
LIN {X 0,Y 199.687,Z 168.608,A -85,B 0,C 180,E1 -21568.134,E2 -21568.134} C_VEL
LIN {X 0,Y 199.677,Z 168.603,A -85,B 0,C 180,E1 -21572.77,E2 -21572.77} C_VEL
LIN {X 0,Y 199.703,Z 168.604,A -85,B 0,C 180,E1 -21577.225,E2 -21577.225} C_VEL
LIN {X 0,Y 199.741,Z 168.604,A -85,B 0,C 180,E1 -21581.798,E2 -21581.798} C_VEL
LIN {X 0,Y 199.803,Z 168.591,A -85,B 0,C 180,E1 -21585.746,E2 -21585.746} C_VEL
LIN {X 0,Y 200.014,Z 168.562,A -85,B 0,C 180,E1 -21589.881,E2 -21589.881} C_VEL
LIN {X 0,Y 199.989,Z 168.527,A -85,B 0,C 180,E1 -21593.948,E2 -21593.948} C_VEL
LIN {X 0,Y 200.275,Z 168.53,A -85,B 0,C 180,E1 -21597.989,E2 -21597.989} C_VEL
LIN {X 0,Y 200.437,Z 168.517,A -85,B 0,C 180,E1 -21600,E2 -21600} C_VEL
LIN {X 0,Y 199.979,Z 168.573,A -85,B 0,C 180,E1 -21604.03,E2 -21604.03} C_VEL
LIN {X 0,Y 200.06,Z 168.562,A -85,B 0,C 180,E1 -21608.078,E2 -21608.078} C_VEL
LIN {X 0,Y 199.855,Z 168.586,A -85,B 0,C 180,E1 -21612.18,E2 -21612.18} C_VEL
LIN {X 0,Y 199.756,Z 168.601,A -85,B 0,C 180,E1 -21616.347,E2 -21616.347} C_VEL
LIN {X 0,Y 199.663,Z 168.614,A -85,B 0,C 180,E1 -21620.609,E2 -21620.609} C_VEL
LIN {X 0,Y 199.656,Z 168.616,A -85,B 0,C 180,E1 -21624.986,E2 -21624.986} C_VEL
LIN {X 0,Y 199.657,Z 168.618,A -85,B 0,C 180,E1 -21629.525,E2 -21629.525} C_VEL
LIN {X 0,Y 199.664,Z 168.62,A -85,B 0,C 180,E1 -21632.357,E2 -21632.357} C_VEL
LIN {X 0,Y 199.616,Z 168.624,A -85,B 0,C 180,E1 -21636.764,E2 -21636.764} C_VEL
LIN {X 0,Y 199.602,Z 168.624,A -85,B 0,C 180,E1 -21639.33,E2 -21639.33} C_VEL
LIN {X 0,Y 199.568,Z 168.628,A -85,B 0,C 180,E1 -21642.312,E2 -21642.312} C_VEL
LIN {X 0,Y 199.626,Z 168.781,A -85,B 0,C 180,E1 -21646.841,E2 -21646.841} C_VEL
LIN {X 0,Y 201.875,Z 177.205,A -85,B 0,C 180,E1 -21651.265,E2 -21651.265} C_VEL
LIN {X 0,Y 204.079,Z 181.606,A -85,B 0,C 180,E1 -21651.902,E2 -21651.902} C_VEL
LIN {X 0,Y 211.052,Z 196.873,A -85,B 0,C 180,E1 -21653.854,E2 -21653.854} C_VEL
LIN {X 0,Y 213.419,Z 202.66,A -85,B 0,C 180,E1 -21654.502,E2 -21654.502} C_VEL
LIN {X 0,Y 214.111,Z 205.68,A -85,B 0,C 180,E1 -21654.74,E2 -21654.74} C_VEL
LIN {X 0,Y 213.755,Z 210.27,A -85,B 0,C 180,E1 -21654.858,E2 -21654.858} C_VEL
LIN {X 0,Y 211.588,Z 219.701,A -85,B 0,C 180,E1 -21654.856,E2 -21654.856} C_VEL
LIN {X 0,Y 211.461,Z 223.79,A -85,B 0,C 180,E1 -21654.996,E2 -21654.996} C_VEL
LIN {X 0,Y 212.835,Z 237.85,A -85,B 0,C 180,E1 -21655.778,E2 -21655.778} C_VEL
LIN {X 0,Y 210.682,Z 286.355,A -85,B 0,C 180,E1 -21657.36,E2 -21657.36} C_VEL
LIN {X 0,Y 209.401,Z 300.007,A -85,B 0,C 180,E1 -21658.162,E2 -21658.162} C_VEL
LIN {X 0,Y 207.603,Z 312.101,A -85,B 0,C 180,E1 -21659.204,E2 -21659.204} C_VEL
LIN {X 0,Y 205.477,Z 323.511,A -85,B 0,C 180,E1 -21660.552,E2 -21660.552} C_VEL
LIN {X 0,Y 202.843,Z 335.253,A -85,B 0,C 180,E1 -21662.395,E2 -21662.395} C_VEL
LIN {X 0,Y 200.21,Z 345.81,A -85,B 0,C 180,E1 -21664.534,E2 -21664.534} C_VEL
LIN {X 0,Y 197.689,Z 355.322,A -85,B 0,C 180,E1 -21666.982,E2 -21666.982} C_VEL
LIN {X 0,Y 195.645,Z 363.121,A -85,B 0,C 180,E1 -21669.5,E2 -21669.5} C_VEL
LIN {X 0,Y 193.6,Z 370.746,A -85,B 0,C 180,E1 -21672.575,E2 -21672.575} C_VEL
LIN {X 0,Y 191.714,Z 377.786,A -85,B 0,C 180,E1 -21676.217,E2 -21676.217} C_VEL
LIN {X 0,Y 190.83,Z 382.452,A -85,B 0,C 180,E1 -21679.391,E2 -21679.391} C_VEL
LIN {X 0,Y 190.385,Z 385.999,A -85,B 0,C 180,E1 -21682.579,E2 -21682.579} C_VEL
LIN {X 0,Y 190.295,Z 388.523,A -85,B 0,C 180,E1 -21685.766,E2 -21685.766} C_VEL
LIN {X 0,Y 190.366,Z 389.686,A -85,B 0,C 180,E1 -21687.886,E2 -21687.886} C_VEL
LIN {X 0,Y 190.493,Z 390.406,A -85,B 0,C 180,E1 -21690.002,E2 -21690.002} C_VEL
LIN {X 0,Y 190.336,Z 390.717,A -85,B 0,C 180,E1 -21692.118,E2 -21692.118} C_VEL
LIN {X 0,Y 190.241,Z 390.639,A -85,B 0,C 180,E1 -21694.239,E2 -21694.239} C_VEL
LIN {X 0,Y 190.241,Z 390.164,A -85,B 0,C 180,E1 -21696.365,E2 -21696.365} C_VEL
LIN {X 0,Y 190.897,Z 387.961,A -85,B 0,C 180,E1 -21700.609,E2 -21700.609} C_VEL
LIN {X 0,Y 191.912,Z 385.235,A -85,B 0,C 180,E1 -21703.772,E2 -21703.772} C_VEL
LIN {X 0,Y 193.555,Z 381.509,A -85,B 0,C 180,E1 -21706.888,E2 -21706.888} C_VEL
LIN {X 0,Y 195.776,Z 376.682,A -85,B 0,C 180,E1 -21709.942,E2 -21709.942} C_VEL
LIN {X 0,Y 198.411,Z 370.609,A -85,B 0,C 180,E1 -21712.934,E2 -21712.934} C_VEL
LIN {X 0,Y 201.56,Z 363.075,A -85,B 0,C 180,E1 -21715.841,E2 -21715.841} C_VEL
LIN {X 0,Y 204.79,Z 355.408,A -85,B 0,C 180,E1 -21718.158,E2 -21718.158} C_VEL
LIN {X 0,Y 208.319,Z 346.107,A -85,B 0,C 180,E1 -21720.403,E2 -21720.403} C_VEL
LIN {X 0,Y 211.816,Z 335.775,A -85,B 0,C 180,E1 -21722.347,E2 -21722.347} C_VEL
LIN {X 0,Y 215.182,Z 324.325,A -85,B 0,C 180,E1 -21724.01,E2 -21724.01} C_VEL
LIN {X 0,Y 218.079,Z 312.36,A -85,B 0,C 180,E1 -21725.316,E2 -21725.316} C_VEL
LIN {X 0,Y 220.485,Z 299.067,A -85,B 0,C 180,E1 -21726.349,E2 -21726.349} C_VEL
LIN {X 0,Y 222.02,Z 285.8,A -85,B 0,C 180,E1 -21727.046,E2 -21727.046} C_VEL
LIN {X 0,Y 224.331,Z 243.35,A -85,B 0,C 180,E1 -21728.345,E2 -21728.345} C_VEL
LIN {X 0,Y 222.449,Z 228.447,A -85,B 0,C 180,E1 -21729.382,E2 -21729.382} C_VEL
LIN {X 0,Y 216.792,Z 215.061,A -85,B 0,C 180,E1 -21731.306,E2 -21731.306} C_VEL
LIN {X 0,Y 210.579,Z 202.287,A -85,B 0,C 180,E1 -21733.526,E2 -21733.526} C_VEL
LIN {X 0,Y 204.537,Z 191.531,A -85,B 0,C 180,E1 -21735.825,E2 -21735.825} C_VEL
LIN {X 0,Y 200.62,Z 185.305,A -85,B 0,C 180,E1 -21737.411,E2 -21737.411} C_VEL
LIN {X 0,Y 197.402,Z 180.16,A -85,B 0,C 180,E1 -21738.803,E2 -21738.803} C_VEL
LIN {X 0,Y 194.481,Z 175.683,A -85,B 0,C 180,E1 -21740.135,E2 -21740.135} C_VEL
LIN {X 0,Y 194.249,Z 175.111,A -85,B 0,C 180,E1 -21740.352,E2 -21740.352} C_VEL
LIN {X 0,Y 192.567,Z 169.498,A -85,B 0,C 180,E1 -21744.753,E2 -21744.753} C_VEL
LIN {X 0,Y 192.574,Z 169.496,A -85,B 0,C 180,E1 -21749.274,E2 -21749.274} C_VEL
LIN {X 0,Y 192.624,Z 169.488,A -85,B 0,C 180,E1 -21751.685,E2 -21751.685} C_VEL
LIN {X 0,Y 192.674,Z 169.482,A -85,B 0,C 180,E1 -21756.345,E2 -21756.345} C_VEL
LIN {X 0,Y 192.698,Z 169.468,A -85,B 0,C 180,E1 -21761.492,E2 -21761.492} C_VEL
LIN {X 0,Y 192.776,Z 169.462,A -85,B 0,C 180,E1 -21767.365,E2 -21767.365} C_VEL
LIN {X 0,Y 193.021,Z 169.423,A -85,B 0,C 180,E1 -21771.626,E2 -21771.626} C_VEL
LIN {X 0,Y 193.211,Z 169.401,A -85,B 0,C 180,E1 -21777.916,E2 -21777.916} C_VEL
LIN {X 0,Y 193.412,Z 169.394,A -85,B 0,C 180,E1 -21780,E2 -21780} C_VEL
LIN {X 0,Y 192.933,Z 169.439,A -85,B 0,C 180,E1 -21784.178,E2 -21784.178} C_VEL
LIN {X 0,Y 193.027,Z 169.423,A -85,B 0,C 180,E1 -21788.374,E2 -21788.374} C_VEL
LIN {X 0,Y 192.791,Z 169.462,A -85,B 0,C 180,E1 -21792.634,E2 -21792.634} C_VEL
LIN {X 0,Y 192.715,Z 169.481,A -85,B 0,C 180,E1 -21796.963,E2 -21796.963} C_VEL
LIN {X 0,Y 192.587,Z 169.493,A -85,B 0,C 180,E1 -21801.403,E2 -21801.403} C_VEL
LIN {X 0,Y 192.639,Z 169.476,A -85,B 0,C 180,E1 -21804.205,E2 -21804.205} C_VEL
LIN {X 0,Y 192.606,Z 169.482,A -85,B 0,C 180,E1 -21808.865,E2 -21808.865} C_VEL
LIN {X 0,Y 192.585,Z 169.494,A -85,B 0,C 180,E1 -21814.289,E2 -21814.289} C_VEL
LIN {X 0,Y 192.591,Z 169.697,A -85,B 0,C 180,E1 -21814.446,E2 -21814.446} C_VEL
LIN {X 0,Y 193.522,Z 172.265,A -85,B 0,C 180,E1 -21814.968,E2 -21814.968} C_VEL
LIN {X 0,Y 195.586,Z 174.457,A -85,B 0,C 180,E1 -21815.884,E2 -21815.884} C_VEL
LIN {X 0,Y 196.317,Z 175.154,A -85,B 0,C 180,E1 -21816.195,E2 -21816.195} C_VEL
LIN {X 0,Y 198.468,Z 178.507,A -85,B 0,C 180,E1 -21817.156,E2 -21817.156} C_VEL
LIN {X 0,Y 199.838,Z 180.041,A -85,B 0,C 180,E1 -21817.715,E2 -21817.715} C_VEL
LIN {X 0,Y 202.613,Z 183.876,A -85,B 0,C 180,E1 -21818.843,E2 -21818.843} C_VEL
LIN {X 0,Y 210.791,Z 195.868,A -85,B 0,C 180,E1 -21821.901,E2 -21821.901} C_VEL
LIN {X 0,Y 218.954,Z 209.472,A -85,B 0,C 180,E1 -21824.655,E2 -21824.655} C_VEL
LIN {X 0,Y 223.548,Z 218.4,A -85,B 0,C 180,E1 -21826.119,E2 -21826.119} C_VEL
LIN {X 0,Y 225.449,Z 223.278,A -85,B 0,C 180,E1 -21826.747,E2 -21826.747} C_VEL
LIN {X 0,Y 222.774,Z 271.139,A -85,B 0,C 180,E1 -21828.215,E2 -21828.215} C_VEL
LIN {X 0,Y 221.207,Z 284.812,A -85,B 0,C 180,E1 -21828.982,E2 -21828.982} C_VEL
LIN {X 0,Y 219.232,Z 296.648,A -85,B 0,C 180,E1 -21829.971,E2 -21829.971} C_VEL
LIN {X 0,Y 216.862,Z 307.78,A -85,B 0,C 180,E1 -21831.243,E2 -21831.243} C_VEL
LIN {X 0,Y 213.921,Z 318.771,A -85,B 0,C 180,E1 -21832.865,E2 -21832.865} C_VEL
LIN {X 0,Y 210.553,Z 329.29,A -85,B 0,C 180,E1 -21834.844,E2 -21834.844} C_VEL
LIN {X 0,Y 207.102,Z 338.737,A -85,B 0,C 180,E1 -21837.113,E2 -21837.113} C_VEL
LIN {X 0,Y 203.723,Z 347.255,A -85,B 0,C 180,E1 -21839.753,E2 -21839.753} C_VEL
LIN {X 0,Y 200.866,Z 353.969,A -85,B 0,C 180,E1 -21842.379,E2 -21842.379} C_VEL
LIN {X 0,Y 197.532,Z 360.895,A -85,B 0,C 180,E1 -21845.846,E2 -21845.846} C_VEL
LIN {X 0,Y 195.215,Z 365.449,A -85,B 0,C 180,E1 -21848.897,E2 -21848.897} C_VEL
LIN {X 0,Y 193.938,Z 367.844,A -85,B 0,C 180,E1 -21850.963,E2 -21850.963} C_VEL
LIN {X 0,Y 192.875,Z 369.795,A -85,B 0,C 180,E1 -21853.05,E2 -21853.05} C_VEL
LIN {X 0,Y 191.954,Z 371.333,A -85,B 0,C 180,E1 -21855.148,E2 -21855.148} C_VEL
LIN {X 0,Y 191.328,Z 372.434,A -85,B 0,C 180,E1 -21857.266,E2 -21857.266} C_VEL
LIN {X 0,Y 190.618,Z 373.409,A -85,B 0,C 180,E1 -21861.517,E2 -21861.517} C_VEL
LIN {X 0,Y 190.506,Z 373.062,A -85,B 0,C 180,E1 -21864.92,E2 -21864.92} C_VEL
LIN {X 0,Y 190.502,Z 371.942,A -85,B 0,C 180,E1 -21867.884,E2 -21867.884} C_VEL
LIN {X 0,Y 190.658,Z 370.66,A -85,B 0,C 180,E1 -21869.998,E2 -21869.998} C_VEL
LIN {X 0,Y 191.161,Z 367.954,A -85,B 0,C 180,E1 -21873.159,E2 -21873.159} C_VEL
LIN {X 0,Y 192.034,Z 364.248,A -85,B 0,C 180,E1 -21876.301,E2 -21876.301} C_VEL
LIN {X 0,Y 193.387,Z 359.429,A -85,B 0,C 180,E1 -21879.41,E2 -21879.41} C_VEL
LIN {X 0,Y 195.1,Z 353.364,A -85,B 0,C 180,E1 -21882.48,E2 -21882.48} C_VEL
LIN {X 0,Y 197.461,Z 345.81,A -85,B 0,C 180,E1 -21885.48,E2 -21885.48} C_VEL
LIN {X 0,Y 200.061,Z 336.329,A -85,B 0,C 180,E1 -21888.429,E2 -21888.429} C_VEL
LIN {X 0,Y 202.588,Z 326.545,A -85,B 0,C 180,E1 -21890.827,E2 -21890.827} C_VEL
LIN {X 0,Y 205.102,Z 315.567,A -85,B 0,C 180,E1 -21892.938,E2 -21892.938} C_VEL
LIN {X 0,Y 207.214,Z 304.814,A -85,B 0,C 180,E1 -21894.547,E2 -21894.547} C_VEL
LIN {X 0,Y 209.044,Z 292.981,A -85,B 0,C 180,E1 -21895.914,E2 -21895.914} C_VEL
LIN {X 0,Y 210.534,Z 280.151,A -85,B 0,C 180,E1 -21896.984,E2 -21896.984} C_VEL
LIN {X 0,Y 211.528,Z 267.476,A -85,B 0,C 180,E1 -21897.65,E2 -21897.65} C_VEL
LIN {X 0,Y 213.965,Z 210.368,A -85,B 0,C 180,E1 -21899.492,E2 -21899.492} C_VEL
LIN {X 0,Y 210.259,Z 201.587,A -85,B 0,C 180,E1 -21900.49,E2 -21900.49} C_VEL
LIN {X 0,Y 202.969,Z 187.431,A -85,B 0,C 180,E1 -21902.464,E2 -21902.464} C_VEL
LIN {X 0,Y 196.478,Z 176.764,A -85,B 0,C 180,E1 -21904.303,E2 -21904.303} C_VEL
LIN {X 0,Y 194.506,Z 173.536,A -85,B 0,C 180,E1 -21904.894,E2 -21904.894} C_VEL
LIN {X 0,Y 193.012,Z 171.162,A -85,B 0,C 180,E1 -21905.35,E2 -21905.35} C_VEL
LIN {X 0,Y 192.595,Z 169.492,A -85,B 0,C 180,E1 -21905.536,E2 -21905.536} C_VEL
LIN {X 0,Y 192.536,Z 169.501,A -85,B 0,C 180,E1 -21909.955,E2 -21909.955} C_VEL
LIN {X 0,Y 192.487,Z 169.506,A -85,B 0,C 180,E1 -21913.922,E2 -21913.922} C_VEL
LIN {X 0,Y 192.508,Z 169.504,A -85,B 0,C 180,E1 -21918.918,E2 -21918.918} C_VEL
LIN {X 0,Y 192.581,Z 169.494,A -85,B 0,C 180,E1 -21923.4,E2 -21923.4} C_VEL
LIN {X 0,Y 192.601,Z 169.486,A -85,B 0,C 180,E1 -21927.058,E2 -21927.058} C_VEL
LIN {X 0,Y 192.654,Z 169.48,A -85,B 0,C 180,E1 -21931.69,E2 -21931.69} C_VEL
LIN {X 0,Y 192.677,Z 169.483,A -85,B 0,C 180,E1 -21936.344,E2 -21936.344} C_VEL
LIN {X 0,Y 192.69,Z 169.484,A -85,B 0,C 180,E1 -21941.487,E2 -21941.487} C_VEL
LIN {X 0,Y 192.729,Z 169.468,A -85,B 0,C 180,E1 -21945.211,E2 -21945.211} C_VEL
LIN {X 0,Y 192.937,Z 169.444,A -85,B 0,C 180,E1 -21949.566,E2 -21949.566} C_VEL
LIN {X 0,Y 192.954,Z 169.402,A -85,B 0,C 180,E1 -21953.727,E2 -21953.727} C_VEL
LIN {X 0,Y 193.219,Z 169.406,A -85,B 0,C 180,E1 -21957.915,E2 -21957.915} C_VEL
LIN {X 0,Y 193.403,Z 169.393,A -85,B 0,C 180,E1 -21960,E2 -21960} C_VEL
LIN {X 0,Y 192.926,Z 169.452,A -85,B 0,C 180,E1 -21964.178,E2 -21964.178} C_VEL
LIN {X 0,Y 193.012,Z 169.44,A -85,B 0,C 180,E1 -21968.375,E2 -21968.375} C_VEL
LIN {X 0,Y 192.782,Z 169.469,A -85,B 0,C 180,E1 -21972.635,E2 -21972.635} C_VEL
LIN {X 0,Y 192.71,Z 169.48,A -85,B 0,C 180,E1 -21976.963,E2 -21976.963} C_VEL
LIN {X 0,Y 192.601,Z 169.496,A -85,B 0,C 180,E1 -21981.401,E2 -21981.401} C_VEL
LIN {X 0,Y 192.639,Z 169.491,A -85,B 0,C 180,E1 -21984.214,E2 -21984.214} C_VEL
LIN {X 0,Y 192.636,Z 169.49,A -85,B 0,C 180,E1 -21988.89,E2 -21988.89} C_VEL
LIN {X 0,Y 192.59,Z 169.499,A -85,B 0,C 180,E1 -21993.187,E2 -21993.187} C_VEL
LIN {X 0,Y 192.545,Z 169.504,A -85,B 0,C 180,E1 -21998.353,E2 -21998.353} C_VEL
LIN {X 0,Y 192.485,Z 169.51,A -85,B 0,C 180,E1 -22003.097,E2 -22003.097} C_VEL
LIN {X 0,Y 192.551,Z 169.513,A -85,B 0,C 180,E1 -22005.59,E2 -22005.59} C_VEL
LIN {X 0,Y 194.516,Z 176.895,A -85,B 0,C 180,E1 -22009.653,E2 -22009.653} C_VEL
LIN {X 0,Y 201.622,Z 191.123,A -85,B 0,C 180,E1 -22011.812,E2 -22011.812} C_VEL
LIN {X 0,Y 207.83,Z 205.624,A -85,B 0,C 180,E1 -22013.621,E2 -22013.621} C_VEL
LIN {X 0,Y 210.132,Z 212.176,A -85,B 0,C 180,E1 -22014.302,E2 -22014.302} C_VEL
LIN {X 0,Y 211.461,Z 223.79,A -85,B 0,C 180,E1 -22014.996,E2 -22014.996} C_VEL
LIN {X 0,Y 211.406,Z 229.637,A -85,B 0,C 180,E1 -22015.217,E2 -22015.217} C_VEL
LIN {X 0,Y 210.329,Z 235.498,A -85,B 0,C 180,E1 -22015.264,E2 -22015.264} C_VEL
LIN {X 0,Y 207.212,Z 247.167,A -85,B 0,C 180,E1 -22015.19,E2 -22015.19} C_VEL
LIN {X 0,Y 206.209,Z 253.099,A -85,B 0,C 180,E1 -22015.254,E2 -22015.254} C_VEL
LIN {X 0,Y 206.092,Z 255.09,A -85,B 0,C 180,E1 -22015.314,E2 -22015.314} C_VEL
LIN {X 0,Y 204.557,Z 286.374,A -85,B 0,C 180,E1 -22016.372,E2 -22016.372} C_VEL
LIN {X 0,Y 203.315,Z 299.472,A -85,B 0,C 180,E1 -22017.164,E2 -22017.164} C_VEL
LIN {X 0,Y 201.339,Z 312.186,A -85,B 0,C 180,E1 -22018.282,E2 -22018.282} C_VEL
LIN {X 0,Y 198.95,Z 324.274,A -85,B 0,C 180,E1 -22019.778,E2 -22019.778} C_VEL
LIN {X 0,Y 196.243,Z 335.815,A -85,B 0,C 180,E1 -22021.675,E2 -22021.675} C_VEL
LIN {X 0,Y 193.5,Z 346.217,A -85,B 0,C 180,E1 -22023.874,E2 -22023.874} C_VEL
LIN {X 0,Y 191.122,Z 354.722,A -85,B 0,C 180,E1 -22026.143,E2 -22026.143} C_VEL
LIN {X 0,Y 188.578,Z 364.073,A -85,B 0,C 180,E1 -22029.318,E2 -22029.318} C_VEL
LIN {X 0,Y 186.494,Z 371.373,A -85,B 0,C 180,E1 -22032.456,E2 -22032.456} C_VEL
LIN {X 0,Y 184.791,Z 377.317,A -85,B 0,C 180,E1 -22035.69,E2 -22035.69} C_VEL
LIN {X 0,Y 183.82,Z 382.015,A -85,B 0,C 180,E1 -22038.981,E2 -22038.981} C_VEL
LIN {X 0,Y 183.325,Z 385.59,A -85,B 0,C 180,E1 -22042.291,E2 -22042.291} C_VEL
LIN {X 0,Y 183.226,Z 388.258,A -85,B 0,C 180,E1 -22045.776,E2 -22045.776} C_VEL
LIN {X 0,Y 183.266,Z 389.328,A -85,B 0,C 180,E1 -22047.804,E2 -22047.804} C_VEL
LIN {X 0,Y 183.408,Z 390.064,A -85,B 0,C 180,E1 -22050.002,E2 -22050.002} C_VEL
LIN {X 0,Y 183.167,Z 390.36,A -85,B 0,C 180,E1 -22053.968,E2 -22053.968} C_VEL
LIN {X 0,Y 183.181,Z 389.865,A -85,B 0,C 180,E1 -22056.611,E2 -22056.611} C_VEL
LIN {X 0,Y 183.889,Z 387.693,A -85,B 0,C 180,E1 -22061.019,E2 -22061.019} C_VEL
LIN {X 0,Y 184.974,Z 384.994,A -85,B 0,C 180,E1 -22064.3,E2 -22064.3} C_VEL
LIN {X 0,Y 186.753,Z 381.298,A -85,B 0,C 180,E1 -22067.523,E2 -22067.523} C_VEL
LIN {X 0,Y 189.102,Z 376.502,A -85,B 0,C 180,E1 -22070.677,E2 -22070.677} C_VEL
LIN {X 0,Y 192.359,Z 369.339,A -85,B 0,C 180,E1 -22074.271,E2 -22074.271} C_VEL
LIN {X 0,Y 195.818,Z 361.563,A -85,B 0,C 180,E1 -22077.234,E2 -22077.234} C_VEL
LIN {X 0,Y 199.969,Z 351.855,A -85,B 0,C 180,E1 -22080.056,E2 -22080.056} C_VEL
